LIN {X 0,Y 523.953,Z 186.844,A -85,B 0,C 180,E1 -4818.69,E2 -4818.69} C_VEL
LIN {X 0,Y 523.915,Z 186.845,A -85,B 0,C 180,E1 -4821.08,E2 -4821.08} C_VEL
LIN {X 0,Y 523.898,Z 186.847,A -85,B 0,C 180,E1 -4823.825,E2 -4823.825} C_VEL
LIN {X 0,Y 523.938,Z 186.841,A -85,B 0,C 180,E1 -4826.635,E2 -4826.635} C_VEL
LIN {X 0,Y 523.953,Z 186.839,A -85,B 0,C 180,E1 -4829.356,E2 -4829.356} C_VEL
LIN {X 0,Y 523.973,Z 186.838,A -85,B 0,C 180,E1 -4832.282,E2 -4832.282} C_VEL
LIN {X 0,Y 523.945,Z 186.843,A -85,B 0,C 180,E1 -4834.581,E2 -4834.581} C_VEL
LIN {X 0,Y 523.916,Z 186.848,A -85,B 0,C 180,E1 -4837.756,E2 -4837.756} C_VEL
LIN {X 0,Y 523.971,Z 186.842,A -85,B 0,C 180,E1 -4840.408,E2 -4840.408} C_VEL
LIN {X 0,Y 523.96,Z 186.838,A -85,B 0,C 180,E1 -4842.837,E2 -4842.837} C_VEL
LIN {X 0,Y 523.974,Z 186.837,A -85,B 0,C 180,E1 -4845.236,E2 -4845.236} C_VEL
LIN {X 0,Y 524.009,Z 186.835,A -85,B 0,C 180,E1 -4848.394,E2 -4848.394} C_VEL
LIN {X 0,Y 524,Z 186.836,A -85,B 0,C 180,E1 -4851.516,E2 -4851.516} C_VEL
LIN {X 0,Y 524.078,Z 186.821,A -85,B 0,C 180,E1 -4854.614,E2 -4854.614} C_VEL
LIN {X 0,Y 524.107,Z 186.827,A -85,B 0,C 180,E1 -4857.695,E2 -4857.695} C_VEL
LIN {X 0,Y 524.12,Z 186.819,A -85,B 0,C 180,E1 -4860.768,E2 -4860.768} C_VEL
LIN {X 0,Y 524.07,Z 186.826,A -85,B 0,C 180,E1 -4863.075,E2 -4863.075} C_VEL
LIN {X 0,Y 524.043,Z 186.829,A -85,B 0,C 180,E1 -4866.159,E2 -4866.159} C_VEL
LIN {X 0,Y 523.996,Z 186.84,A -85,B 0,C 180,E1 -4869.262,E2 -4869.262} C_VEL
LIN {X 0,Y 524,Z 186.835,A -85,B 0,C 180,E1 -4871.74,E2 -4871.74} C_VEL
LIN {X 0,Y 523.991,Z 186.841,A -85,B 0,C 180,E1 -4875.053,E2 -4875.053} C_VEL
LIN {X 0,Y 523.962,Z 186.839,A -85,B 0,C 180,E1 -4877.969,E2 -4877.969} C_VEL
LIN {X 0,Y 523.97,Z 186.836,A -85,B 0,C 180,E1 -4880.41,E2 -4880.41} C_VEL
LIN {X 0,Y 523.909,Z 186.851,A -85,B 0,C 180,E1 -4882.894,E2 -4882.894} C_VEL
LIN {X 0,Y 523.951,Z 186.843,A -85,B 0,C 180,E1 -4885.419,E2 -4885.419} C_VEL
LIN {X 0,Y 523.966,Z 186.832,A -85,B 0,C 180,E1 -4887.999,E2 -4887.999} C_VEL
LIN {X 0,Y 523.943,Z 186.846,A -85,B 0,C 180,E1 -4890.855,E2 -4890.855} C_VEL
LIN {X 0,Y 523.96,Z 186.835,A -85,B 0,C 180,E1 -4893.735,E2 -4893.735} C_VEL
LIN {X 0,Y 523.922,Z 186.845,A -85,B 0,C 180,E1 -4896.405,E2 -4896.405} C_VEL
LIN {X 0,Y 523.919,Z 186.842,A -85,B 0,C 180,E1 -4899.085,E2 -4899.085} C_VEL
LIN {X 0,Y 523.951,Z 186.843,A -85,B 0,C 180,E1 -4902.119,E2 -4902.119} C_VEL
LIN {X 0,Y 523.946,Z 186.841,A -85,B 0,C 180,E1 -4905.31,E2 -4905.31} C_VEL
LIN {X 0,Y 523.917,Z 186.845,A -85,B 0,C 180,E1 -4906.914,E2 -4906.914} C_VEL
LIN {X 0,Y 523.253,Z 186.926,A -85,B 0,C 180,E1 -4907.556,E2 -4907.556} C_VEL
LIN {X 0,Y 520.411,Z 187.287,A -85,B 0,C 180,E1 -4908.597,E2 -4908.597} C_VEL
LIN {X 0,Y 518.006,Z 187.591,A -85,B 0,C 180,E1 -4909.436,E2 -4909.436} C_VEL
LIN {X 0,Y 516.969,Z 187.718,A -85,B 0,C 180,E1 -4910.084,E2 -4910.084} C_VEL
LIN {X 0,Y 516.881,Z 187.727,A -85,B 0,C 180,E1 -4910.303,E2 -4910.303} C_VEL
LIN {X 0,Y 516.88,Z 187.72,A -85,B 0,C 180,E1 -4913.343,E2 -4913.343} C_VEL
LIN {X 0,Y 516.912,Z 187.715,A -85,B 0,C 180,E1 -4916.121,E2 -4916.121} C_VEL
LIN {X 0,Y 516.893,Z 187.722,A -85,B 0,C 180,E1 -4918.936,E2 -4918.936} C_VEL
LIN {X 0,Y 516.864,Z 187.729,A -85,B 0,C 180,E1 -4921.582,E2 -4921.582} C_VEL
LIN {X 0,Y 516.931,Z 187.951,A -85,B 0,C 180,E1 -4922.974,E2 -4922.974} C_VEL
LIN {X 0,Y 519.733,Z 200.118,A -85,B 0,C 180,E1 -4924.958,E2 -4924.958} C_VEL
LIN {X 0,Y 519.555,Z 209.088,A -85,B 0,C 180,E1 -4926.27,E2 -4926.27} C_VEL
LIN {X 0,Y 518.755,Z 230.793,A -85,B 0,C 180,E1 -4929.375,E2 -4929.375} C_VEL
LIN {X 0,Y 518.392,Z 244.374,A -85,B 0,C 180,E1 -4931.264,E2 -4931.264} C_VEL
LIN {X 0,Y 520.841,Z 257.475,A -85,B 0,C 180,E1 -4931.568,E2 -4931.568} C_VEL
LIN {X 0,Y 520.186,Z 383.262,A -85,B 0,C 180,E1 -4933.29,E2 -4933.29} C_VEL
LIN {X 0,Y 519.944,Z 397.944,A -85,B 0,C 180,E1 -4933.652,E2 -4933.652} C_VEL
LIN {X 0,Y 519.646,Z 411.088,A -85,B 0,C 180,E1 -4934.131,E2 -4934.131} C_VEL
LIN {X 0,Y 519.251,Z 424.666,A -85,B 0,C 180,E1 -4934.797,E2 -4934.797} C_VEL
LIN {X 0,Y 518.721,Z 437.26,A -85,B 0,C 180,E1 -4935.584,E2 -4935.584} C_VEL
LIN {X 0,Y 518.328,Z 448.694,A -85,B 0,C 180,E1 -4936.474,E2 -4936.474} C_VEL
LIN {X 0,Y 517.874,Z 459.183,A -85,B 0,C 180,E1 -4937.459,E2 -4937.459} C_VEL
LIN {X 0,Y 517.46,Z 469.589,A -85,B 0,C 180,E1 -4938.642,E2 -4938.642} C_VEL
LIN {X 0,Y 517.091,Z 478.189,A -85,B 0,C 180,E1 -4939.823,E2 -4939.823} C_VEL
LIN {X 0,Y 516.781,Z 486.445,A -85,B 0,C 180,E1 -4941.199,E2 -4941.199} C_VEL
LIN {X 0,Y 516.571,Z 493.107,A -85,B 0,C 180,E1 -4942.574,E2 -4942.574} C_VEL
LIN {X 0,Y 516.504,Z 497.705,A -85,B 0,C 180,E1 -4943.75,E2 -4943.75} C_VEL
LIN {X 0,Y 516.312,Z 502.484,A -85,B 0,C 180,E1 -4945.315,E2 -4945.315} C_VEL
LIN {X 0,Y 516.357,Z 505.807,A -85,B 0,C 180,E1 -4946.879,E2 -4946.879} C_VEL
LIN {X 0,Y 516.191,Z 507.794,A -85,B 0,C 180,E1 -4948.439,E2 -4948.439} C_VEL
LIN {X 0,Y 516.166,Z 508.48,A -85,B 0,C 180,E1 -4950,E2 -4950} C_VEL
LIN {X 0,Y 516.189,Z 507.88,A -85,B 0,C 180,E1 -4951.56,E2 -4951.56} C_VEL
LIN {X 0,Y 516.356,Z 505.975,A -85,B 0,C 180,E1 -4953.121,E2 -4953.121} C_VEL
LIN {X 0,Y 516.311,Z 502.723,A -85,B 0,C 180,E1 -4954.684,E2 -4954.684} C_VEL
LIN {X 0,Y 516.502,Z 498.019,A -85,B 0,C 180,E1 -4956.249,E2 -4956.249} C_VEL
LIN {X 0,Y 516.599,Z 491.746,A -85,B 0,C 180,E1 -4957.819,E2 -4957.819} C_VEL
LIN {X 0,Y 516.828,Z 484.765,A -85,B 0,C 180,E1 -4959.194,E2 -4959.194} C_VEL
LIN {X 0,Y 517.185,Z 476.143,A -85,B 0,C 180,E1 -4960.57,E2 -4960.57} C_VEL
LIN {X 0,Y 517.563,Z 467.127,A -85,B 0,C 180,E1 -4961.752,E2 -4961.752} C_VEL
LIN {X 0,Y 517.889,Z 458.139,A -85,B 0,C 180,E1 -4962.739,E2 -4962.739} C_VEL
LIN {X 0,Y 518.339,Z 447.432,A -85,B 0,C 180,E1 -4963.725,E2 -4963.725} C_VEL
LIN {X 0,Y 518.789,Z 435.723,A -85,B 0,C 180,E1 -4964.614,E2 -4964.614} C_VEL
LIN {X 0,Y 519.285,Z 422.762,A -85,B 0,C 180,E1 -4965.402,E2 -4965.402} C_VEL
LIN {X 0,Y 519.719,Z 409.76,A -85,B 0,C 180,E1 -4966.014,E2 -4966.014} C_VEL
LIN {X 0,Y 519.993,Z 396.813,A -85,B 0,C 180,E1 -4966.472,E2 -4966.472} C_VEL
LIN {X 0,Y 520.192,Z 382.646,A -85,B 0,C 180,E1 -4966.81,E2 -4966.81} C_VEL
LIN {X 0,Y 520.805,Z 261.865,A -85,B 0,C 180,E1 -4968.461,E2 -4968.461} C_VEL
LIN {X 0,Y 520.611,Z 255.697,A -85,B 0,C 180,E1 -4968.554,E2 -4968.554} C_VEL
LIN {X 0,Y 518.438,Z 244.638,A -85,B 0,C 180,E1 -4968.809,E2 -4968.809} C_VEL
LIN {X 0,Y 518.502,Z 238.716,A -85,B 0,C 180,E1 -4969.601,E2 -4969.601} C_VEL
LIN {X 0,Y 519.191,Z 218.613,A -85,B 0,C 180,E1 -4972.453,E2 -4972.453} C_VEL
LIN {X 0,Y 519.801,Z 200.601,A -85,B 0,C 180,E1 -4975.058,E2 -4975.058} C_VEL
LIN {X 0,Y 516.902,Z 187.815,A -85,B 0,C 180,E1 -4977.163,E2 -4977.163} C_VEL
LIN {X 0,Y 516.89,Z 187.718,A -85,B 0,C 180,E1 -4980.203,E2 -4980.203} C_VEL
LIN {X 0,Y 516.894,Z 187.715,A -85,B 0,C 180,E1 -4982.946,E2 -4982.946} C_VEL
LIN {X 0,Y 516.887,Z 187.726,A -85,B 0,C 180,E1 -4985.778,E2 -4985.778} C_VEL
LIN {X 0,Y 516.878,Z 187.721,A -85,B 0,C 180,E1 -4988.715,E2 -4988.715} C_VEL
LIN {X 0,Y 516.911,Z 187.72,A -85,B 0,C 180,E1 -4991.774,E2 -4991.774} C_VEL
LIN {X 0,Y 516.919,Z 187.719,A -85,B 0,C 180,E1 -4995.009,E2 -4995.009} C_VEL
LIN {X 0,Y 516.913,Z 187.718,A -85,B 0,C 180,E1 -4998.398,E2 -4998.398} C_VEL
LIN {X 0,Y 516.877,Z 187.724,A -85,B 0,C 180,E1 -5001.283,E2 -5001.283} C_VEL
LIN {X 0,Y 516.886,Z 187.718,A -85,B 0,C 180,E1 -5004.221,E2 -5004.221} C_VEL
LIN {X 0,Y 516.891,Z 187.722,A -85,B 0,C 180,E1 -5007.053,E2 -5007.053} C_VEL
LIN {X 0,Y 516.896,Z 187.716,A -85,B 0,C 180,E1 -5009.796,E2 -5009.796} C_VEL
LIN {X 0,Y 516.923,Z 187.71,A -85,B 0,C 180,E1 -5012.467,E2 -5012.467} C_VEL
LIN {X 0,Y 516.904,Z 187.725,A -85,B 0,C 180,E1 -5015.071,E2 -5015.071} C_VEL
LIN {X 0,Y 516.863,Z 187.724,A -85,B 0,C 180,E1 -5017.621,E2 -5017.621} C_VEL
LIN {X 0,Y 516.926,Z 187.713,A -85,B 0,C 180,E1 -5020.129,E2 -5020.129} C_VEL
LIN {X 0,Y 516.925,Z 187.721,A -85,B 0,C 180,E1 -5022.596,E2 -5022.596} C_VEL
LIN {X 0,Y 516.935,Z 187.719,A -85,B 0,C 180,E1 -5025.03,E2 -5025.03} C_VEL
LIN {X 0,Y 516.958,Z 187.712,A -85,B 0,C 180,E1 -5028.233,E2 -5028.233} C_VEL
LIN {X 0,Y 516.963,Z 187.71,A -85,B 0,C 180,E1 -5031.399,E2 -5031.399} C_VEL
LIN {X 0,Y 517.003,Z 187.705,A -85,B 0,C 180,E1 -5033.757,E2 -5033.757} C_VEL
LIN {X 0,Y 517.077,Z 187.695,A -85,B 0,C 180,E1 -5037.663,E2 -5037.663} C_VEL
LIN {X 0,Y 517.087,Z 187.695,A -85,B 0,C 180,E1 -5040.779,E2 -5040.779} C_VEL
LIN {X 0,Y 517.008,Z 187.705,A -85,B 0,C 180,E1 -5043.117,E2 -5043.117} C_VEL
LIN {X 0,Y 517.004,Z 187.71,A -85,B 0,C 180,E1 -5046.243,E2 -5046.243} C_VEL
LIN {X 0,Y 516.947,Z 187.711,A -85,B 0,C 180,E1 -5049.389,E2 -5049.389} C_VEL
LIN {X 0,Y 516.944,Z 187.717,A -85,B 0,C 180,E1 -5051.807,E2 -5051.807} C_VEL
LIN {X 0,Y 516.936,Z 187.713,A -85,B 0,C 180,E1 -5055.147,E2 -5055.147} C_VEL
LIN {X 0,Y 516.918,Z 187.721,A -85,B 0,C 180,E1 -5058.222,E2 -5058.222} C_VEL
LIN {X 0,Y 516.905,Z 187.717,A -85,B 0,C 180,E1 -5060.702,E2 -5060.702} C_VEL
LIN {X 0,Y 516.904,Z 187.721,A -85,B 0,C 180,E1 -5064.072,E2 -5064.072} C_VEL
LIN {X 0,Y 516.921,Z 187.706,A -85,B 0,C 180,E1 -5066.658,E2 -5066.658} C_VEL
LIN {X 0,Y 516.903,Z 187.724,A -85,B 0,C 180,E1 -5069.524,E2 -5069.524} C_VEL
LIN {X 0,Y 516.891,Z 187.711,A -85,B 0,C 180,E1 -5072.544,E2 -5072.544} C_VEL
LIN {X 0,Y 516.874,Z 187.728,A -85,B 0,C 180,E1 -5075.332,E2 -5075.332} C_VEL
LIN {X 0,Y 516.875,Z 187.722,A -85,B 0,C 180,E1 -5077.944,E2 -5077.944} C_VEL
LIN {X 0,Y 516.877,Z 187.723,A -85,B 0,C 180,E1 -5080.742,E2 -5080.742} C_VEL
LIN {X 0,Y 516.876,Z 187.721,A -85,B 0,C 180,E1 -5082.832,E2 -5082.832} C_VEL
LIN {X 0,Y 516.889,Z 187.725,A -85,B 0,C 180,E1 -5085.007,E2 -5085.007} C_VEL
LIN {X 0,Y 516.908,Z 187.717,A -85,B 0,C 180,E1 -5088.399,E2 -5088.399} C_VEL
LIN {X 0,Y 516.873,Z 187.719,A -85,B 0,C 180,E1 -5091.284,E2 -5091.284} C_VEL
LIN {X 0,Y 516.866,Z 187.719,A -85,B 0,C 180,E1 -5094.22,E2 -5094.22} C_VEL
LIN {X 0,Y 516.877,Z 187.725,A -85,B 0,C 180,E1 -5097.053,E2 -5097.053} C_VEL
LIN {X 0,Y 516.857,Z 187.678,A -85,B 0,C 180,E1 -5099.795,E2 -5099.795} C_VEL
LIN {X 0,Y 516.926,Z 187.879,A -85,B 0,C 180,E1 -5101.392,E2 -5101.392} C_VEL
LIN {X 0,Y 520.508,Z 201.805,A -85,B 0,C 180,E1 -5103.314,E2 -5103.314} C_VEL
LIN {X 0,Y 520.721,Z 205.507,A -85,B 0,C 180,E1 -5103.768,E2 -5103.768} C_VEL
LIN {X 0,Y 519.625,Z 234.25,A -85,B 0,C 180,E1 -5107.118,E2 -5107.118} C_VEL
LIN {X 0,Y 519.292,Z 245.134,A -85,B 0,C 180,E1 -5108.345,E2 -5108.345} C_VEL
LIN {X 0,Y 521.579,Z 259.663,A -85,B 0,C 180,E1 -5108.666,E2 -5108.666} C_VEL
LIN {X 0,Y 520.369,Z 411.25,A -85,B 0,C 180,E1 -5110.871,E2 -5110.871} C_VEL
LIN {X 0,Y 520.061,Z 427.069,A -85,B 0,C 180,E1 -5111.265,E2 -5111.265} C_VEL
LIN {X 0,Y 519.736,Z 441.63,A -85,B 0,C 180,E1 -5111.784,E2 -5111.784} C_VEL
LIN {X 0,Y 519.225,Z 456.376,A -85,B 0,C 180,E1 -5112.473,E2 -5112.473} C_VEL
LIN {X 0,Y 518.806,Z 469.902,A -85,B 0,C 180,E1 -5113.27,E2 -5113.27} C_VEL
LIN {X 0,Y 518.308,Z 483.631,A -85,B 0,C 180,E1 -5114.265,E2 -5114.265} C_VEL
LIN {X 0,Y 517.839,Z 496.096,A -85,B 0,C 180,E1 -5115.359,E2 -5115.359} C_VEL
LIN {X 0,Y 517.44,Z 506.568,A -85,B 0,C 180,E1 -5116.45,E2 -5116.45} C_VEL
LIN {X 0,Y 517.045,Z 517.733,A -85,B 0,C 180,E1 -5117.838,E2 -5117.838} C_VEL
LIN {X 0,Y 516.819,Z 526.971,A -85,B 0,C 180,E1 -5119.224,E2 -5119.224} C_VEL
LIN {X 0,Y 516.55,Z 534.62,A -85,B 0,C 180,E1 -5120.604,E2 -5120.604} C_VEL
LIN {X 0,Y 516.443,Z 541.759,A -85,B 0,C 180,E1 -5122.179,E2 -5122.179} C_VEL
LIN {X 0,Y 516.36,Z 547.363,A -85,B 0,C 180,E1 -5123.749,E2 -5123.749} C_VEL
LIN {X 0,Y 516.374,Z 549.645,A -85,B 0,C 180,E1 -5124.533,E2 -5124.533} C_VEL
LIN {X 0,Y 516.307,Z 553.23,A -85,B 0,C 180,E1 -5126.098,E2 -5126.098} C_VEL
LIN {X 0,Y 516.258,Z 555.585,A -85,B 0,C 180,E1 -5127.66,E2 -5127.66} C_VEL
LIN {X 0,Y 516.157,Z 556.764,A -85,B 0,C 180,E1 -5129.22,E2 -5129.22} C_VEL
LIN {X 0,Y 516.158,Z 556.763,A -85,B 0,C 180,E1 -5130.78,E2 -5130.78} C_VEL
LIN {X 0,Y 516.258,Z 555.58,A -85,B 0,C 180,E1 -5132.341,E2 -5132.341} C_VEL
LIN {X 0,Y 516.307,Z 553.225,A -85,B 0,C 180,E1 -5133.903,E2 -5133.903} C_VEL
LIN {X 0,Y 516.374,Z 549.645,A -85,B 0,C 180,E1 -5135.467,E2 -5135.467} C_VEL
LIN {X 0,Y 516.396,Z 544.743,A -85,B 0,C 180,E1 -5137.036,E2 -5137.036} C_VEL
LIN {X 0,Y 516.514,Z 538.389,A -85,B 0,C 180,E1 -5138.608,E2 -5138.608} C_VEL
LIN {X 0,Y 516.699,Z 530.4,A -85,B 0,C 180,E1 -5140.185,E2 -5140.185} C_VEL
LIN {X 0,Y 516.915,Z 522.234,A -85,B 0,C 180,E1 -5141.517,E2 -5141.517} C_VEL
LIN {X 0,Y 517.199,Z 513.193,A -85,B 0,C 180,E1 -5142.757,E2 -5142.757} C_VEL
LIN {X 0,Y 517.58,Z 502.929,A -85,B 0,C 180,E1 -5143.947,E2 -5143.947} C_VEL
LIN {X 0,Y 518,Z 491.056,A -85,B 0,C 180,E1 -5145.106,E2 -5145.106} C_VEL
LIN {X 0,Y 518.467,Z 478.419,A -85,B 0,C 180,E1 -5146.134,E2 -5146.134} C_VEL
LIN {X 0,Y 518.9,Z 465.073,A -85,B 0,C 180,E1 -5147.031,E2 -5147.031} C_VEL
LIN {X 0,Y 519.391,Z 451.396,A -85,B 0,C 180,E1 -5147.776,E2 -5147.776} C_VEL
LIN {X 0,Y 519.85,Z 436.725,A -85,B 0,C 180,E1 -5148.405,E2 -5148.405} C_VEL
LIN {X 0,Y 520.174,Z 422.03,A -85,B 0,C 180,E1 -5148.876,E2 -5148.876} C_VEL
LIN {X 0,Y 520.43,Z 406.572,A -85,B 0,C 180,E1 -5149.21,E2 -5149.21} C_VEL
LIN {X 0,Y 521.524,Z 258.21,A -85,B 0,C 180,E1 -5151.357,E2 -5151.357} C_VEL
LIN {X 0,Y 519.277,Z 244.941,A -85,B 0,C 180,E1 -5151.668,E2 -5151.668} C_VEL
LIN {X 0,Y 520.013,Z 223.524,A -85,B 0,C 180,E1 -5154.131,E2 -5154.131} C_VEL
LIN {X 0,Y 520.77,Z 203.694,A -85,B 0,C 180,E1 -5156.446,E2 -5156.446} C_VEL
LIN {X 0,Y 519.83,Z 199.121,A -85,B 0,C 180,E1 -5157.044,E2 -5157.044} C_VEL
LIN {X 0,Y 516.929,Z 187.877,A -85,B 0,C 180,E1 -5158.608,E2 -5158.608} C_VEL
LIN {X 0,Y 516.885,Z 187.686,A -85,B 0,C 180,E1 -5161.11,E2 -5161.11} C_VEL
LIN {X 0,Y 516.884,Z 187.722,A -85,B 0,C 180,E1 -5163.962,E2 -5163.962} C_VEL
LIN {X 0,Y 516.875,Z 187.724,A -85,B 0,C 180,E1 -5166.746,E2 -5166.746} C_VEL
LIN {X 0,Y 516.869,Z 187.707,A -85,B 0,C 180,E1 -5169.722,E2 -5169.722} C_VEL
LIN {X 0,Y 516.91,Z 187.717,A -85,B 0,C 180,E1 -5171.775,E2 -5171.775} C_VEL
LIN {X 0,Y 516.893,Z 187.725,A -85,B 0,C 180,E1 -5175.007,E2 -5175.007} C_VEL
LIN {X 0,Y 516.911,Z 187.718,A -85,B 0,C 180,E1 -5178.399,E2 -5178.399} C_VEL
LIN {X 0,Y 516.878,Z 187.72,A -85,B 0,C 180,E1 -5181.284,E2 -5181.284} C_VEL
LIN {X 0,Y 516.868,Z 187.726,A -85,B 0,C 180,E1 -5184.22,E2 -5184.22} C_VEL
LIN {X 0,Y 516.892,Z 187.713,A -85,B 0,C 180,E1 -5187.053,E2 -5187.053} C_VEL
LIN {X 0,Y 516.888,Z 187.721,A -85,B 0,C 180,E1 -5189.796,E2 -5189.796} C_VEL
LIN {X 0,Y 516.923,Z 187.712,A -85,B 0,C 180,E1 -5192.467,E2 -5192.467} C_VEL
LIN {X 0,Y 516.873,Z 187.72,A -85,B 0,C 180,E1 -5195.07,E2 -5195.07} C_VEL
LIN {X 0,Y 516.865,Z 187.725,A -85,B 0,C 180,E1 -5197.621,E2 -5197.621} C_VEL
LIN {X 0,Y 516.928,Z 187.723,A -85,B 0,C 180,E1 -5200.13,E2 -5200.13} C_VEL
LIN {X 0,Y 516.924,Z 187.716,A -85,B 0,C 180,E1 -5202.596,E2 -5202.596} C_VEL
LIN {X 0,Y 516.939,Z 187.713,A -85,B 0,C 180,E1 -5205.03,E2 -5205.03} C_VEL
LIN {X 0,Y 516.963,Z 187.715,A -85,B 0,C 180,E1 -5208.234,E2 -5208.234} C_VEL
LIN {X 0,Y 516.965,Z 187.711,A -85,B 0,C 180,E1 -5211.4,E2 -5211.4} C_VEL
LIN {X 0,Y 517.007,Z 187.71,A -85,B 0,C 180,E1 -5213.757,E2 -5213.757} C_VEL
LIN {X 0,Y 517.08,Z 187.702,A -85,B 0,C 180,E1 -5217.663,E2 -5217.663} C_VEL
LIN {X 0,Y 517.09,Z 187.695,A -85,B 0,C 180,E1 -5220.779,E2 -5220.779} C_VEL
LIN {X 0,Y 517.011,Z 187.705,A -85,B 0,C 180,E1 -5223.117,E2 -5223.117} C_VEL
LIN {X 0,Y 517.007,Z 187.705,A -85,B 0,C 180,E1 -5226.243,E2 -5226.243} C_VEL
LIN {X 0,Y 516.951,Z 187.72,A -85,B 0,C 180,E1 -5229.389,E2 -5229.389} C_VEL
LIN {X 0,Y 516.949,Z 187.713,A -85,B 0,C 180,E1 -5231.807,E2 -5231.807} C_VEL
LIN {X 0,Y 516.942,Z 187.72,A -85,B 0,C 180,E1 -5235.147,E2 -5235.147} C_VEL
LIN {X 0,Y 516.923,Z 187.716,A -85,B 0,C 180,E1 -5238.222,E2 -5238.222} C_VEL
LIN {X 0,Y 516.91,Z 187.717,A -85,B 0,C 180,E1 -5240.702,E2 -5240.702} C_VEL
LIN {X 0,Y 516.901,Z 187.716,A -85,B 0,C 180,E1 -5244.073,E2 -5244.073} C_VEL
LIN {X 0,Y 516.922,Z 187.72,A -85,B 0,C 180,E1 -5246.658,E2 -5246.658} C_VEL
LIN {X 0,Y 516.909,Z 187.715,A -85,B 0,C 180,E1 -5249.524,E2 -5249.524} C_VEL
LIN {X 0,Y 516.894,Z 187.724,A -85,B 0,C 180,E1 -5252.544,E2 -5252.544} C_VEL
LIN {X 0,Y 516.882,Z 187.719,A -85,B 0,C 180,E1 -5255.333,E2 -5255.333} C_VEL
LIN {X 0,Y 516.88,Z 187.722,A -85,B 0,C 180,E1 -5257.943,E2 -5257.943} C_VEL
LIN {X 0,Y 516.882,Z 187.724,A -85,B 0,C 180,E1 -5260.742,E2 -5260.742} C_VEL
LIN {X 0,Y 516.882,Z 187.724,A -85,B 0,C 180,E1 -5262.832,E2 -5262.832} C_VEL
LIN {X 0,Y 516.923,Z 187.719,A -85,B 0,C 180,E1 -5265.01,E2 -5265.01} C_VEL
LIN {X 0,Y 516.916,Z 187.72,A -85,B 0,C 180,E1 -5268.399,E2 -5268.399} C_VEL
LIN {X 0,Y 516.881,Z 187.727,A -85,B 0,C 180,E1 -5270.303,E2 -5270.303} C_VEL
LIN {X 0,Y 516.21,Z 187.807,A -85,B 0,C 180,E1 -5270.953,E2 -5270.953} C_VEL
LIN {X 0,Y 513.363,Z 188.163,A -85,B 0,C 180,E1 -5272.009,E2 -5272.009} C_VEL
LIN {X 0,Y 510.954,Z 188.46,A -85,B 0,C 180,E1 -5272.859,E2 -5272.859} C_VEL
LIN {X 0,Y 509.913,Z 188.588,A -85,B 0,C 180,E1 -5273.516,E2 -5273.516} C_VEL
LIN {X 0,Y 509.824,Z 188.6,A -85,B 0,C 180,E1 -5273.738,E2 -5273.738} C_VEL
LIN {X 0,Y 509.862,Z 188.589,A -85,B 0,C 180,E1 -5276.539,E2 -5276.539} C_VEL
LIN {X 0,Y 509.847,Z 188.599,A -85,B 0,C 180,E1 -5279.334,E2 -5279.334} C_VEL
LIN {X 0,Y 509.871,Z 188.59,A -85,B 0,C 180,E1 -5282.499,E2 -5282.499} C_VEL
LIN {X 0,Y 509.907,Z 189.025,A -85,B 0,C 180,E1 -5282.724,E2 -5282.724} C_VEL
LIN {X 0,Y 512.941,Z 201.979,A -85,B 0,C 180,E1 -5284.866,E2 -5284.866} C_VEL
LIN {X 0,Y 512.535,Z 214.705,A -85,B 0,C 180,E1 -5286.74,E2 -5286.74} C_VEL
LIN {X 0,Y 511.72,Z 236.742,A -85,B 0,C 180,E1 -5289.919,E2 -5289.919} C_VEL
LIN {X 0,Y 511.525,Z 244.588,A -85,B 0,C 180,E1 -5290.994,E2 -5290.994} C_VEL
LIN {X 0,Y 514.172,Z 258.182,A -85,B 0,C 180,E1 -5291.307,E2 -5291.307} C_VEL
LIN {X 0,Y 513.489,Z 384.022,A -85,B 0,C 180,E1 -5293.04,E2 -5293.04} C_VEL
LIN {X 0,Y 513.247,Z 398.289,A -85,B 0,C 180,E1 -5293.399,E2 -5293.399} C_VEL
LIN {X 0,Y 512.891,Z 412.102,A -85,B 0,C 180,E1 -5293.912,E2 -5293.912} C_VEL
LIN {X 0,Y 512.552,Z 423.868,A -85,B 0,C 180,E1 -5294.492,E2 -5294.492} C_VEL
LIN {X 0,Y 511.992,Z 436.682,A -85,B 0,C 180,E1 -5295.289,E2 -5295.289} C_VEL
LIN {X 0,Y 511.511,Z 448.28,A -85,B 0,C 180,E1 -5296.188,E2 -5296.188} C_VEL
LIN {X 0,Y 510.987,Z 459.837,A -85,B 0,C 180,E1 -5297.287,E2 -5297.287} C_VEL
LIN {X 0,Y 510.52,Z 470.169,A -85,B 0,C 180,E1 -5298.486,E2 -5298.486} C_VEL
LIN {X 0,Y 510.13,Z 478.708,A -85,B 0,C 180,E1 -5299.683,E2 -5299.683} C_VEL
LIN {X 0,Y 509.781,Z 486.911,A -85,B 0,C 180,E1 -5301.077,E2 -5301.077} C_VEL
LIN {X 0,Y 509.546,Z 493.532,A -85,B 0,C 180,E1 -5302.471,E2 -5302.471} C_VEL
LIN {X 0,Y 509.413,Z 499.453,A -85,B 0,C 180,E1 -5304.061,E2 -5304.061} C_VEL
LIN {X 0,Y 509.231,Z 502.855,A -85,B 0,C 180,E1 -5305.25,E2 -5305.25} C_VEL
LIN {X 0,Y 509.281,Z 506.157,A -85,B 0,C 180,E1 -5306.835,E2 -5306.835} C_VEL
LIN {X 0,Y 509.111,Z 508.132,A -85,B 0,C 180,E1 -5308.418,E2 -5308.418} C_VEL
LIN {X 0,Y 509.076,Z 508.812,A -85,B 0,C 180,E1 -5310,E2 -5310} C_VEL
LIN {X 0,Y 509.11,Z 508.215,A -85,B 0,C 180,E1 -5311.582,E2 -5311.582} C_VEL
LIN {X 0,Y 509.266,Z 506.323,A -85,B 0,C 180,E1 -5313.164,E2 -5313.164} C_VEL
LIN {X 0,Y 509.23,Z 503.09,A -85,B 0,C 180,E1 -5314.75,E2 -5314.75} C_VEL
LIN {X 0,Y 509.465,Z 498.412,A -85,B 0,C 180,E1 -5316.336,E2 -5316.336} C_VEL
LIN {X 0,Y 509.58,Z 492.172,A -85,B 0,C 180,E1 -5317.927,E2 -5317.927} C_VEL
LIN {X 0,Y 509.836,Z 485.229,A -85,B 0,C 180,E1 -5319.321,E2 -5319.321} C_VEL
LIN {X 0,Y 510.223,Z 476.657,A -85,B 0,C 180,E1 -5320.716,E2 -5320.716} C_VEL
LIN {X 0,Y 510.639,Z 467.7,A -85,B 0,C 180,E1 -5321.914,E2 -5321.914} C_VEL
LIN {X 0,Y 511.121,Z 456.852,A -85,B 0,C 180,E1 -5323.113,E2 -5323.113} C_VEL
LIN {X 0,Y 511.602,Z 445.802,A -85,B 0,C 180,E1 -5324.113,E2 -5324.113} C_VEL
LIN {X 0,Y 512.136,Z 433.594,A -85,B 0,C 180,E1 -5325.011,E2 -5325.011} C_VEL
LIN {X 0,Y 512.571,Z 421.835,A -85,B 0,C 180,E1 -5325.711,E2 -5325.711} C_VEL
LIN {X 0,Y 513.004,Z 409.13,A -85,B 0,C 180,E1 -5326.303,E2 -5326.303} C_VEL
LIN {X 0,Y 513.297,Z 395.96,A -85,B 0,C 180,E1 -5326.761,E2 -5326.761} C_VEL
LIN {X 0,Y 513.509,Z 381.878,A -85,B 0,C 180,E1 -5327.087,E2 -5327.087} C_VEL
LIN {X 0,Y 514.144,Z 258.405,A -85,B 0,C 180,E1 -5328.78,E2 -5328.78} C_VEL
LIN {X 0,Y 511.545,Z 244.541,A -85,B 0,C 180,E1 -5329.099,E2 -5329.099} C_VEL
LIN {X 0,Y 511.938,Z 230.922,A -85,B 0,C 180,E1 -5331.009,E2 -5331.009} C_VEL
LIN {X 0,Y 512.728,Z 209.821,A -85,B 0,C 180,E1 -5334.065,E2 -5334.065} C_VEL
LIN {X 0,Y 512.877,Z 201.786,A -85,B 0,C 180,E1 -5335.257,E2 -5335.257} C_VEL
LIN {X 0,Y 509.882,Z 188.697,A -85,B 0,C 180,E1 -5337.444,E2 -5337.444} C_VEL
LIN {X 0,Y 509.844,Z 188.599,A -85,B 0,C 180,E1 -5340.665,E2 -5340.665} C_VEL
LIN {X 0,Y 509.859,Z 188.589,A -85,B 0,C 180,E1 -5343.46,E2 -5343.46} C_VEL
LIN {X 0,Y 509.833,Z 188.599,A -85,B 0,C 180,E1 -5346.352,E2 -5346.352} C_VEL
LIN {X 0,Y 509.831,Z 188.602,A -85,B 0,C 180,E1 -5349.47,E2 -5349.47} C_VEL
LIN {X 0,Y 509.831,Z 188.596,A -85,B 0,C 180,E1 -5352.489,E2 -5352.489} C_VEL
LIN {X 0,Y 509.853,Z 188.6,A -85,B 0,C 180,E1 -5355.331,E2 -5355.331} C_VEL
LIN {X 0,Y 509.855,Z 188.597,A -85,B 0,C 180,E1 -5358.574,E2 -5358.574} C_VEL
LIN {X 0,Y 509.846,Z 188.601,A -85,B 0,C 180,E1 -5361.786,E2 -5361.786} C_VEL
LIN {X 0,Y 509.841,Z 188.596,A -85,B 0,C 180,E1 -5364.623,E2 -5364.623} C_VEL
LIN {X 0,Y 509.858,Z 188.601,A -85,B 0,C 180,E1 -5367.48,E2 -5367.48} C_VEL
LIN {X 0,Y 509.876,Z 188.589,A -85,B 0,C 180,E1 -5370.268,E2 -5370.268} C_VEL
LIN {X 0,Y 509.88,Z 188.593,A -85,B 0,C 180,E1 -5372.944,E2 -5372.944} C_VEL
LIN {X 0,Y 509.863,Z 188.595,A -85,B 0,C 180,E1 -5375.574,E2 -5375.574} C_VEL
LIN {X 0,Y 509.844,Z 188.603,A -85,B 0,C 180,E1 -5378.998,E2 -5378.998} C_VEL
LIN {X 0,Y 509.882,Z 188.593,A -85,B 0,C 180,E1 -5381.999,E2 -5381.999} C_VEL
LIN {X 0,Y 509.903,Z 188.595,A -85,B 0,C 180,E1 -5384.818,E2 -5384.818} C_VEL
LIN {X 0,Y 509.894,Z 188.59,A -85,B 0,C 180,E1 -5388.123,E2 -5388.123} C_VEL
LIN {X 0,Y 509.909,Z 188.589,A -85,B 0,C 180,E1 -5391.28,E2 -5391.28} C_VEL
LIN {X 0,Y 509.971,Z 188.581,A -85,B 0,C 180,E1 -5393.67,E2 -5393.67} C_VEL
LIN {X 0,Y 510.048,Z 188.57,A -85,B 0,C 180,E1 -5397.631,E2 -5397.631} C_VEL
LIN {X 0,Y 510.057,Z 188.57,A -85,B 0,C 180,E1 -5400.789,E2 -5400.789} C_VEL
LIN {X 0,Y 509.95,Z 188.584,A -85,B 0,C 180,E1 -5403.16,E2 -5403.16} C_VEL
LIN {X 0,Y 509.972,Z 188.587,A -85,B 0,C 180,E1 -5406.33,E2 -5406.33} C_VEL
LIN {X 0,Y 509.909,Z 188.589,A -85,B 0,C 180,E1 -5408.72,E2 -5408.72} C_VEL
LIN {X 0,Y 509.896,Z 188.597,A -85,B 0,C 180,E1 -5411.932,E2 -5411.932} C_VEL
LIN {X 0,Y 509.886,Z 188.592,A -85,B 0,C 180,E1 -5415.242,E2 -5415.242} C_VEL
LIN {X 0,Y 509.881,Z 188.597,A -85,B 0,C 180,E1 -5418.001,E2 -5418.001} C_VEL
LIN {X 0,Y 509.843,Z 188.596,A -85,B 0,C 180,E1 -5421.002,E2 -5421.002} C_VEL
LIN {X 0,Y 509.863,Z 188.594,A -85,B 0,C 180,E1 -5424.426,E2 -5424.426} C_VEL
LIN {X 0,Y 509.88,Z 188.584,A -85,B 0,C 180,E1 -5427.056,E2 -5427.056} C_VEL
LIN {X 0,Y 509.85,Z 188.604,A -85,B 0,C 180,E1 -5429.751,E2 -5429.751} C_VEL
LIN {X 0,Y 509.868,Z 188.586,A -85,B 0,C 180,E1 -5432.775,E2 -5432.775} C_VEL
LIN {X 0,Y 509.834,Z 188.605,A -85,B 0,C 180,E1 -5435.581,E2 -5435.581} C_VEL
LIN {X 0,Y 509.844,Z 188.595,A -85,B 0,C 180,E1 -5438.338,E2 -5438.338} C_VEL
LIN {X 0,Y 509.849,Z 188.599,A -85,B 0,C 180,E1 -5441.426,E2 -5441.426} C_VEL
LIN {X 0,Y 509.833,Z 188.601,A -85,B 0,C 180,E1 -5444.67,E2 -5444.67} C_VEL
LIN {X 0,Y 509.85,Z 188.596,A -85,B 0,C 180,E1 -5448.104,E2 -5448.104} C_VEL
LIN {X 0,Y 509.833,Z 188.585,A -85,B 0,C 180,E1 -5450.647,E2 -5450.647} C_VEL
LIN {X 0,Y 509.82,Z 188.598,A -85,B 0,C 180,E1 -5453.647,E2 -5453.647} C_VEL
LIN {X 0,Y 509.837,Z 188.603,A -85,B 0,C 180,E1 -5456.538,E2 -5456.538} C_VEL
LIN {X 0,Y 509.828,Z 188.556,A -85,B 0,C 180,E1 -5459.334,E2 -5459.334} C_VEL
LIN {X 0,Y 509.901,Z 188.758,A -85,B 0,C 180,E1 -5461.088,E2 -5461.088} C_VEL
LIN {X 0,Y 513.696,Z 203.561,A -85,B 0,C 180,E1 -5463.162,E2 -5463.162} C_VEL
LIN {X 0,Y 514.036,Z 205.372,A -85,B 0,C 180,E1 -5463.4,E2 -5463.4} C_VEL
LIN {X 0,Y 512.857,Z 234.031,A -85,B 0,C 180,E1 -5466.792,E2 -5466.792} C_VEL
LIN {X 0,Y 512.462,Z 245.285,A -85,B 0,C 180,E1 -5468.069,E2 -5468.069} C_VEL
LIN {X 0,Y 514.912,Z 260.394,A -85,B 0,C 180,E1 -5468.409,E2 -5468.409} C_VEL
LIN {X 0,Y 513.575,Z 411.141,A -85,B 0,C 180,E1 -5470.646,E2 -5470.646} C_VEL
LIN {X 0,Y 513.254,Z 426.906,A -85,B 0,C 180,E1 -5471.047,E2 -5471.047} C_VEL
LIN {X 0,Y 512.869,Z 441.694,A -85,B 0,C 180,E1 -5471.584,E2 -5471.584} C_VEL
LIN {X 0,Y 512.379,Z 455.418,A -85,B 0,C 180,E1 -5472.231,E2 -5472.231} C_VEL
LIN {X 0,Y 511.89,Z 469.037,A -85,B 0,C 180,E1 -5473.038,E2 -5473.038} C_VEL
LIN {X 0,Y 511.353,Z 482.887,A -85,B 0,C 180,E1 -5474.046,E2 -5474.046} C_VEL
LIN {X 0,Y 510.861,Z 495.432,A -85,B 0,C 180,E1 -5475.154,E2 -5475.154} C_VEL
LIN {X 0,Y 510.381,Z 507.693,A -85,B 0,C 180,E1 -5476.462,E2 -5476.462} C_VEL
LIN {X 0,Y 510.001,Z 517.196,A -85,B 0,C 180,E1 -5477.667,E2 -5477.667} C_VEL
LIN {X 0,Y 509.743,Z 526.491,A -85,B 0,C 180,E1 -5479.072,E2 -5479.072} C_VEL
LIN {X 0,Y 509.476,Z 534.184,A -85,B 0,C 180,E1 -5480.472,E2 -5480.472} C_VEL
LIN {X 0,Y 509.361,Z 541.357,A -85,B 0,C 180,E1 -5482.07,E2 -5482.07} C_VEL
LIN {X 0,Y 509.265,Z 546.985,A -85,B 0,C 180,E1 -5483.662,E2 -5483.662} C_VEL
LIN {X 0,Y 509.158,Z 551.233,A -85,B 0,C 180,E1 -5485.25,E2 -5485.25} C_VEL
LIN {X 0,Y 509.188,Z 554.212,A -85,B 0,C 180,E1 -5486.835,E2 -5486.835} C_VEL
LIN {X 0,Y 509.11,Z 555.983,A -85,B 0,C 180,E1 -5488.418,E2 -5488.418} C_VEL
LIN {X 0,Y 509.064,Z 556.587,A -85,B 0,C 180,E1 -5490,E2 -5490} C_VEL
LIN {X 0,Y 509.11,Z 555.98,A -85,B 0,C 180,E1 -5491.582,E2 -5491.582} C_VEL
LIN {X 0,Y 509.188,Z 554.206,A -85,B 0,C 180,E1 -5493.165,E2 -5493.165} C_VEL
LIN {X 0,Y 509.158,Z 551.229,A -85,B 0,C 180,E1 -5494.751,E2 -5494.751} C_VEL
LIN {X 0,Y 509.306,Z 546.99,A -85,B 0,C 180,E1 -5496.338,E2 -5496.338} C_VEL
LIN {X 0,Y 509.362,Z 541.355,A -85,B 0,C 180,E1 -5497.931,E2 -5497.931} C_VEL
LIN {X 0,Y 509.476,Z 534.175,A -85,B 0,C 180,E1 -5499.528,E2 -5499.528} C_VEL
LIN {X 0,Y 509.739,Z 526.484,A -85,B 0,C 180,E1 -5500.928,E2 -5500.928} C_VEL
LIN {X 0,Y 510.006,Z 517.194,A -85,B 0,C 180,E1 -5502.333,E2 -5502.333} C_VEL
LIN {X 0,Y 510.442,Z 505.946,A -85,B 0,C 180,E1 -5503.739,E2 -5503.739} C_VEL
LIN {X 0,Y 510.918,Z 494.363,A -85,B 0,C 180,E1 -5504.947,E2 -5504.947} C_VEL
LIN {X 0,Y 511.359,Z 482.891,A -85,B 0,C 180,E1 -5505.955,E2 -5505.955} C_VEL
LIN {X 0,Y 511.865,Z 469.024,A -85,B 0,C 180,E1 -5506.964,E2 -5506.964} C_VEL
LIN {X 0,Y 512.407,Z 454.405,A -85,B 0,C 180,E1 -5507.82,E2 -5507.82} C_VEL
LIN {X 0,Y 512.931,Z 439.537,A -85,B 0,C 180,E1 -5508.504,E2 -5508.504} C_VEL
LIN {X 0,Y 513.294,Z 424.558,A -85,B 0,C 180,E1 -5509.024,E2 -5509.024} C_VEL
LIN {X 0,Y 513.601,Z 409.813,A -85,B 0,C 180,E1 -5509.38,E2 -5509.38} C_VEL
LIN {X 0,Y 514.903,Z 259.98,A -85,B 0,C 180,E1 -5511.597,E2 -5511.597} C_VEL
LIN {X 0,Y 512.447,Z 244.964,A -85,B 0,C 180,E1 -5511.948,E2 -5511.948} C_VEL
LIN {X 0,Y 513.202,Z 225.177,A -85,B 0,C 180,E1 -5514.257,E2 -5514.257} C_VEL
LIN {X 0,Y 514.006,Z 205.361,A -85,B 0,C 180,E1 -5516.602,E2 -5516.602} C_VEL
LIN {X 0,Y 510.66,Z 191.731,A -85,B 0,C 180,E1 -5518.465,E2 -5518.465} C_VEL
LIN {X 0,Y 509.891,Z 188.72,A -85,B 0,C 180,E1 -5518.928,E2 -5518.928} C_VEL
LIN {X 0,Y 509.816,Z 188.577,A -85,B 0,C 180,E1 -5521.59,E2 -5521.59} C_VEL
LIN {X 0,Y 509.836,Z 188.597,A -85,B 0,C 180,E1 -5524.414,E2 -5524.414} C_VEL
LIN {X 0,Y 509.814,Z 188.605,A -85,B 0,C 180,E1 -5527.341,E2 -5527.341} C_VEL
LIN {X 0,Y 509.836,Z 188.585,A -85,B 0,C 180,E1 -5530.382,E2 -5530.382} C_VEL
LIN {X 0,Y 509.82,Z 188.605,A -85,B 0,C 180,E1 -5533.062,E2 -5533.062} C_VEL
LIN {X 0,Y 509.82,Z 188.601,A -85,B 0,C 180,E1 -5535.793,E2 -5535.793} C_VEL
LIN {X 0,Y 509.853,Z 188.598,A -85,B 0,C 180,E1 -5538.574,E2 -5538.574} C_VEL
LIN {X 0,Y 509.848,Z 188.595,A -85,B 0,C 180,E1 -5541.786,E2 -5541.786} C_VEL
LIN {X 0,Y 509.828,Z 188.607,A -85,B 0,C 180,E1 -5544.622,E2 -5544.622} C_VEL
LIN {X 0,Y 509.858,Z 188.587,A -85,B 0,C 180,E1 -5547.481,E2 -5547.481} C_VEL
LIN {X 0,Y 509.855,Z 188.603,A -85,B 0,C 180,E1 -5550.274,E2 -5550.274} C_VEL
LIN {X 0,Y 509.881,Z 188.583,A -85,B 0,C 180,E1 -5552.944,E2 -5552.944} C_VEL
LIN {X 0,Y 509.848,Z 188.596,A -85,B 0,C 180,E1 -5555.573,E2 -5555.573} C_VEL
LIN {X 0,Y 509.819,Z 188.606,A -85,B 0,C 180,E1 -5558.149,E2 -5558.149} C_VEL
LIN {X 0,Y 509.86,Z 188.597,A -85,B 0,C 180,E1 -5560.682,E2 -5560.682} C_VEL
LIN {X 0,Y 509.878,Z 188.592,A -85,B 0,C 180,E1 -5563.175,E2 -5563.175} C_VEL
LIN {X 0,Y 509.861,Z 188.599,A -85,B 0,C 180,E1 -5565.634,E2 -5565.634} C_VEL
LIN {X 0,Y 509.91,Z 188.589,A -85,B 0,C 180,E1 -5568.875,E2 -5568.875} C_VEL
LIN {X 0,Y 509.948,Z 188.589,A -85,B 0,C 180,E1 -5572.079,E2 -5572.079} C_VEL
LIN {X 0,Y 509.978,Z 188.578,A -85,B 0,C 180,E1 -5574.464,E2 -5574.464} C_VEL
LIN {X 0,Y 510.051,Z 188.578,A -85,B 0,C 180,E1 -5577.631,E2 -5577.631} C_VEL
LIN {X 0,Y 510.061,Z 188.57,A -85,B 0,C 180,E1 -5580.79,E2 -5580.79} C_VEL
LIN {X 0,Y 509.953,Z 188.585,A -85,B 0,C 180,E1 -5583.16,E2 -5583.16} C_VEL
LIN {X 0,Y 509.975,Z 188.58,A -85,B 0,C 180,E1 -5586.33,E2 -5586.33} C_VEL
LIN {X 0,Y 509.913,Z 188.588,A -85,B 0,C 180,E1 -5588.72,E2 -5588.72} C_VEL
LIN {X 0,Y 509.902,Z 188.589,A -85,B 0,C 180,E1 -5591.932,E2 -5591.932} C_VEL
LIN {X 0,Y 509.892,Z 188.597,A -85,B 0,C 180,E1 -5595.242,E2 -5595.242} C_VEL
LIN {X 0,Y 509.88,Z 188.593,A -85,B 0,C 180,E1 -5597.999,E2 -5597.999} C_VEL
LIN {X 0,Y 509.848,Z 188.601,A -85,B 0,C 180,E1 -5601.002,E2 -5601.002} C_VEL
LIN {X 0,Y 509.862,Z 188.595,A -85,B 0,C 180,E1 -5604.427,E2 -5604.427} C_VEL
LIN {X 0,Y 509.882,Z 188.594,A -85,B 0,C 180,E1 -5607.056,E2 -5607.056} C_VEL
LIN {X 0,Y 509.856,Z 188.592,A -85,B 0,C 180,E1 -5609.751,E2 -5609.751} C_VEL
LIN {X 0,Y 509.872,Z 188.601,A -85,B 0,C 180,E1 -5612.774,E2 -5612.774} C_VEL
LIN {X 0,Y 509.842,Z 188.595,A -85,B 0,C 180,E1 -5615.581,E2 -5615.581} C_VEL
LIN {X 0,Y 509.849,Z 188.601,A -85,B 0,C 180,E1 -5618.338,E2 -5618.338} C_VEL
LIN {X 0,Y 509.854,Z 188.597,A -85,B 0,C 180,E1 -5621.426,E2 -5621.426} C_VEL
LIN {X 0,Y 509.857,Z 188.599,A -85,B 0,C 180,E1 -5624.668,E2 -5624.668} C_VEL
LIN {X 0,Y 509.858,Z 188.596,A -85,B 0,C 180,E1 -5628.103,E2 -5628.103} C_VEL
LIN {X 0,Y 509.846,Z 188.6,A -85,B 0,C 180,E1 -5630.648,E2 -5630.648} C_VEL
LIN {X 0,Y 509.824,Z 188.6,A -85,B 0,C 180,E1 -5633.738,E2 -5633.738} C_VEL
LIN {X 0,Y 509.158,Z 188.691,A -85,B 0,C 180,E1 -5634.398,E2 -5634.398} C_VEL
LIN {X 0,Y 506.344,Z 189.035,A -85,B 0,C 180,E1 -5635.47,E2 -5635.47} C_VEL
LIN {X 0,Y 503.955,Z 189.326,A -85,B 0,C 180,E1 -5636.333,E2 -5636.333} C_VEL
LIN {X 0,Y 502.907,Z 189.454,A -85,B 0,C 180,E1 -5637,E2 -5637} C_VEL
LIN {X 0,Y 502.809,Z 189.466,A -85,B 0,C 180,E1 -5637.225,E2 -5637.225} C_VEL
LIN {X 0,Y 502.816,Z 189.468,A -85,B 0,C 180,E1 -5640.065,E2 -5640.065} C_VEL
LIN {X 0,Y 502.875,Z 189.695,A -85,B 0,C 180,E1 -5642.395,E2 -5642.395} C_VEL
LIN {X 0,Y 506.093,Z 203.615,A -85,B 0,C 180,E1 -5644.733,E2 -5644.733} C_VEL
LIN {X 0,Y 505.9,Z 212.213,A -85,B 0,C 180,E1 -5646.025,E2 -5646.025} C_VEL
LIN {X 0,Y 504.962,Z 234.156,A -85,B 0,C 180,E1 -5649.238,E2 -5649.238} C_VEL
LIN {X 0,Y 504.625,Z 244.422,A -85,B 0,C 180,E1 -5650.69,E2 -5650.69} C_VEL
LIN {X 0,Y 507.536,Z 259.583,A -85,B 0,C 180,E1 -5651.05,E2 -5651.05} C_VEL
LIN {X 0,Y 506.816,Z 384.647,A -85,B 0,C 180,E1 -5652.784,E2 -5652.784} C_VEL
LIN {X 0,Y 506.549,Z 398.703,A -85,B 0,C 180,E1 -5653.142,E2 -5653.142} C_VEL
LIN {X 0,Y 506.193,Z 412.044,A -85,B 0,C 180,E1 -5653.64,E2 -5653.64} C_VEL
LIN {X 0,Y 505.857,Z 423.042,A -85,B 0,C 180,E1 -5654.178,E2 -5654.178} C_VEL
LIN {X 0,Y 505.246,Z 436.105,A -85,B 0,C 180,E1 -5654.985,E2 -5654.985} C_VEL
LIN {X 0,Y 504.718,Z 447.863,A -85,B 0,C 180,E1 -5655.896,E2 -5655.896} C_VEL
LIN {X 0,Y 504.153,Z 458.589,A -85,B 0,C 180,E1 -5656.907,E2 -5656.907} C_VEL
LIN {X 0,Y 503.688,Z 469.169,A -85,B 0,C 180,E1 -5658.123,E2 -5658.123} C_VEL
LIN {X 0,Y 503.23,Z 477.924,A -85,B 0,C 180,E1 -5659.336,E2 -5659.336} C_VEL
LIN {X 0,Y 502.805,Z 486.311,A -85,B 0,C 180,E1 -5660.75,E2 -5660.75} C_VEL
LIN {X 0,Y 502.584,Z 492.213,A -85,B 0,C 180,E1 -5661.961,E2 -5661.961} C_VEL
LIN {X 0,Y 502.402,Z 498.508,A -85,B 0,C 180,E1 -5663.574,E2 -5663.574} C_VEL
LIN {X 0,Y 502.152,Z 503.231,A -85,B 0,C 180,E1 -5665.183,E2 -5665.183} C_VEL
LIN {X 0,Y 502.194,Z 506.51,A -85,B 0,C 180,E1 -5666.791,E2 -5666.791} C_VEL
LIN {X 0,Y 502.035,Z 508.47,A -85,B 0,C 180,E1 -5668.395,E2 -5668.395} C_VEL
LIN {X 0,Y 501.99,Z 509.145,A -85,B 0,C 180,E1 -5670,E2 -5670} C_VEL
LIN {X 0,Y 502.034,Z 508.551,A -85,B 0,C 180,E1 -5671.604,E2 -5671.604} C_VEL
LIN {X 0,Y 502.181,Z 506.672,A -85,B 0,C 180,E1 -5673.209,E2 -5673.209} C_VEL
LIN {X 0,Y 502.151,Z 503.461,A -85,B 0,C 180,E1 -5674.817,E2 -5674.817} C_VEL
LIN {X 0,Y 502.402,Z 498.811,A -85,B 0,C 180,E1 -5676.425,E2 -5676.425} C_VEL
LIN {X 0,Y 502.544,Z 492.607,A -85,B 0,C 180,E1 -5678.039,E2 -5678.039} C_VEL
LIN {X 0,Y 502.841,Z 485.707,A -85,B 0,C 180,E1 -5679.452,E2 -5679.452} C_VEL
LIN {X 0,Y 503.268,Z 477.187,A -85,B 0,C 180,E1 -5680.866,E2 -5680.866} C_VEL
LIN {X 0,Y 503.748,Z 467.136,A -85,B 0,C 180,E1 -5682.226,E2 -5682.226} C_VEL
LIN {X 0,Y 504.288,Z 456.486,A -85,B 0,C 180,E1 -5683.396,E2 -5683.396} C_VEL
LIN {X 0,Y 504.838,Z 445.293,A -85,B 0,C 180,E1 -5684.409,E2 -5684.409} C_VEL
LIN {X 0,Y 505.421,Z 432.895,A -85,B 0,C 180,E1 -5685.319,E2 -5685.319} C_VEL
LIN {X 0,Y 505.829,Z 420.865,A -85,B 0,C 180,E1 -5686.03,E2 -5686.03} C_VEL
LIN {X 0,Y 506.346,Z 406.743,A -85,B 0,C 180,E1 -5686.666,E2 -5686.666} C_VEL
LIN {X 0,Y 506.663,Z 392.828,A -85,B 0,C 180,E1 -5687.117,E2 -5687.117} C_VEL
LIN {X 0,Y 506.863,Z 379.391,A -85,B 0,C 180,E1 -5687.396,E2 -5687.396} C_VEL
LIN {X 0,Y 507.466,Z 260.171,A -85,B 0,C 180,E1 -5689.034,E2 -5689.034} C_VEL
LIN {X 0,Y 507.019,Z 256.502,A -85,B 0,C 180,E1 -5689.105,E2 -5689.105} C_VEL
LIN {X 0,Y 504.637,Z 244.319,A -85,B 0,C 180,E1 -5689.407,E2 -5689.407} C_VEL
LIN {X 0,Y 505.335,Z 224.469,A -85,B 0,C 180,E1 -5692.27,E2 -5692.27} C_VEL
LIN {X 0,Y 506.158,Z 205.703,A -85,B 0,C 180,E1 -5695.035,E2 -5695.035} C_VEL
LIN {X 0,Y 505.882,Z 202.678,A -85,B 0,C 180,E1 -5695.509,E2 -5695.509} C_VEL
LIN {X 0,Y 502.84,Z 189.563,A -85,B 0,C 180,E1 -5697.748,E2 -5697.748} C_VEL
LIN {X 0,Y 502.808,Z 189.47,A -85,B 0,C 180,E1 -5700.21,E2 -5700.21} C_VEL
LIN {X 0,Y 502.83,Z 189.464,A -85,B 0,C 180,E1 -5703.03,E2 -5703.03} C_VEL
LIN {X 0,Y 502.78,Z 189.481,A -85,B 0,C 180,E1 -5705.95,E2 -5705.95} C_VEL
LIN {X 0,Y 502.799,Z 189.476,A -85,B 0,C 180,E1 -5708.975,E2 -5708.975} C_VEL
LIN {X 0,Y 502.793,Z 189.475,A -85,B 0,C 180,E1 -5712.138,E2 -5712.138} C_VEL
LIN {X 0,Y 502.797,Z 189.477,A -85,B 0,C 180,E1 -5715.468,E2 -5715.468} C_VEL
LIN {X 0,Y 502.817,Z 189.476,A -85,B 0,C 180,E1 -5718.934,E2 -5718.934} C_VEL
LIN {X 0,Y 502.789,Z 189.478,A -85,B 0,C 180,E1 -5722.045,E2 -5722.045} C_VEL
LIN {X 0,Y 502.805,Z 189.473,A -85,B 0,C 180,E1 -5725.034,E2 -5725.034} C_VEL
LIN {X 0,Y 502.779,Z 189.479,A -85,B 0,C 180,E1 -5727.915,E2 -5727.915} C_VEL
LIN {X 0,Y 502.834,Z 189.469,A -85,B 0,C 180,E1 -5730.713,E2 -5730.713} C_VEL
LIN {X 0,Y 502.856,Z 189.471,A -85,B 0,C 180,E1 -5733.439,E2 -5733.439} C_VEL
LIN {X 0,Y 502.785,Z 189.475,A -85,B 0,C 180,E1 -5736.086,E2 -5736.086} C_VEL
LIN {X 0,Y 502.777,Z 189.483,A -85,B 0,C 180,E1 -5738.688,E2 -5738.688} C_VEL
LIN {X 0,Y 502.824,Z 189.476,A -85,B 0,C 180,E1 -5741.248,E2 -5741.248} C_VEL
LIN {X 0,Y 502.817,Z 189.47,A -85,B 0,C 180,E1 -5743.767,E2 -5743.767} C_VEL
LIN {X 0,Y 502.829,Z 189.474,A -85,B 0,C 180,E1 -5746.254,E2 -5746.254} C_VEL
LIN {X 0,Y 502.87,Z 189.47,A -85,B 0,C 180,E1 -5748.717,E2 -5748.717} C_VEL
LIN {X 0,Y 502.895,Z 189.463,A -85,B 0,C 180,E1 -5751.966,E2 -5751.966} C_VEL
LIN {X 0,Y 502.932,Z 189.464,A -85,B 0,C 180,E1 -5754.386,E2 -5754.386} C_VEL
LIN {X 0,Y 503.018,Z 189.446,A -85,B 0,C 180,E1 -5757.598,E2 -5757.598} C_VEL
LIN {X 0,Y 503.019,Z 189.451,A -85,B 0,C 180,E1 -5760,E2 -5760} C_VEL
LIN {X 0,Y 503.017,Z 189.454,A -85,B 0,C 180,E1 -5762.402,E2 -5762.402} C_VEL
LIN {X 0,Y 502.931,Z 189.456,A -85,B 0,C 180,E1 -5765.613,E2 -5765.613} C_VEL
LIN {X 0,Y 502.894,Z 189.469,A -85,B 0,C 180,E1 -5768.033,E2 -5768.033} C_VEL
LIN {X 0,Y 502.869,Z 189.466,A -85,B 0,C 180,E1 -5771.283,E2 -5771.283} C_VEL
LIN {X 0,Y 502.838,Z 189.471,A -85,B 0,C 180,E1 -5774.571,E2 -5774.571} C_VEL
LIN {X 0,Y 502.854,Z 189.472,A -85,B 0,C 180,E1 -5777.907,E2 -5777.907} C_VEL
LIN {X 0,Y 502.821,Z 189.472,A -85,B 0,C 180,E1 -5780.536,E2 -5780.536} C_VEL
LIN {X 0,Y 502.787,Z 189.477,A -85,B 0,C 180,E1 -5783.041,E2 -5783.041} C_VEL
LIN {X 0,Y 502.835,Z 189.468,A -85,B 0,C 180,E1 -5785.676,E2 -5785.676} C_VEL
LIN {X 0,Y 502.832,Z 189.471,A -85,B 0,C 180,E1 -5788.373,E2 -5788.373} C_VEL
LIN {X 0,Y 502.787,Z 189.478,A -85,B 0,C 180,E1 -5791.499,E2 -5791.499} C_VEL
LIN {X 0,Y 502.799,Z 189.475,A -85,B 0,C 180,E1 -5794.445,E2 -5794.445} C_VEL
LIN {X 0,Y 502.774,Z 189.479,A -85,B 0,C 180,E1 -5797.179,E2 -5797.179} C_VEL
LIN {X 0,Y 502.782,Z 189.479,A -85,B 0,C 180,E1 -5800.016,E2 -5800.016} C_VEL
LIN {X 0,Y 502.797,Z 189.472,A -85,B 0,C 180,E1 -5802.2,E2 -5802.2} C_VEL
LIN {X 0,Y 502.78,Z 189.479,A -85,B 0,C 180,E1 -5805.471,E2 -5805.471} C_VEL
LIN {X 0,Y 502.815,Z 189.469,A -85,B 0,C 180,E1 -5808.935,E2 -5808.935} C_VEL
LIN {X 0,Y 502.788,Z 189.478,A -85,B 0,C 180,E1 -5812.047,E2 -5812.047} C_VEL
LIN {X 0,Y 502.791,Z 189.468,A -85,B 0,C 180,E1 -5815.034,E2 -5815.034} C_VEL
LIN {X 0,Y 502.778,Z 189.468,A -85,B 0,C 180,E1 -5817.916,E2 -5817.916} C_VEL
LIN {X 0,Y 502.866,Z 189.629,A -85,B 0,C 180,E1 -5820.77,E2 -5820.77} C_VEL
LIN {X 0,Y 507.002,Z 205.751,A -85,B 0,C 180,E1 -5823.066,E2 -5823.066} C_VEL
LIN {X 0,Y 507.225,Z 208.84,A -85,B 0,C 180,E1 -5823.459,E2 -5823.459} C_VEL
LIN {X 0,Y 505.864,Z 239.295,A -85,B 0,C 180,E1 -5827.108,E2 -5827.108} C_VEL
LIN {X 0,Y 505.607,Z 245.069,A -85,B 0,C 180,E1 -5827.769,E2 -5827.769} C_VEL
LIN {X 0,Y 508.251,Z 261.328,A -85,B 0,C 180,E1 -5828.149,E2 -5828.149} C_VEL
LIN {X 0,Y 506.789,Z 410.468,A -85,B 0,C 180,E1 -5830.402,E2 -5830.402} C_VEL
LIN {X 0,Y 506.447,Z 425.937,A -85,B 0,C 180,E1 -5830.796,E2 -5830.796} C_VEL
LIN {X 0,Y 505.995,Z 441.585,A -85,B 0,C 180,E1 -5831.37,E2 -5831.37} C_VEL
LIN {X 0,Y 505.448,Z 456.286,A -85,B 0,C 180,E1 -5832.084,E2 -5832.084} C_VEL
LIN {X 0,Y 504.931,Z 469.705,A -85,B 0,C 180,E1 -5832.901,E2 -5832.901} C_VEL
LIN {X 0,Y 504.359,Z 483.631,A -85,B 0,C 180,E1 -5833.946,E2 -5833.946} C_VEL
LIN {X 0,Y 503.851,Z 495.774,A -85,B 0,C 180,E1 -5835.046,E2 -5835.046} C_VEL
LIN {X 0,Y 503.366,Z 507.096,A -85,B 0,C 180,E1 -5836.27,E2 -5836.27} C_VEL
LIN {X 0,Y 502.973,Z 516.639,A -85,B 0,C 180,E1 -5837.492,E2 -5837.492} C_VEL
LIN {X 0,Y 502.682,Z 525.985,A -85,B 0,C 180,E1 -5838.917,E2 -5838.917} C_VEL
LIN {X 0,Y 502.406,Z 533.724,A -85,B 0,C 180,E1 -5840.337,E2 -5840.337} C_VEL
LIN {X 0,Y 502.276,Z 540.939,A -85,B 0,C 180,E1 -5841.957,E2 -5841.957} C_VEL
LIN {X 0,Y 502.184,Z 546.601,A -85,B 0,C 180,E1 -5843.572,E2 -5843.572} C_VEL
LIN {X 0,Y 502.081,Z 550.873,A -85,B 0,C 180,E1 -5845.183,E2 -5845.183} C_VEL
LIN {X 0,Y 502.107,Z 553.868,A -85,B 0,C 180,E1 -5846.791,E2 -5846.791} C_VEL
LIN {X 0,Y 502.034,Z 555.648,A -85,B 0,C 180,E1 -5848.396,E2 -5848.396} C_VEL
LIN {X 0,Y 501.979,Z 556.255,A -85,B 0,C 180,E1 -5850,E2 -5850} C_VEL
LIN {X 0,Y 502.034,Z 555.646,A -85,B 0,C 180,E1 -5851.605,E2 -5851.605} C_VEL
LIN {X 0,Y 502.107,Z 553.862,A -85,B 0,C 180,E1 -5853.21,E2 -5853.21} C_VEL
LIN {X 0,Y 502.081,Z 550.87,A -85,B 0,C 180,E1 -5854.818,E2 -5854.818} C_VEL
LIN {X 0,Y 502.233,Z 546.606,A -85,B 0,C 180,E1 -5856.428,E2 -5856.428} C_VEL
LIN {X 0,Y 502.276,Z 540.938,A -85,B 0,C 180,E1 -5858.044,E2 -5858.044} C_VEL
LIN {X 0,Y 502.406,Z 533.715,A -85,B 0,C 180,E1 -5859.664,E2 -5859.664} C_VEL
LIN {X 0,Y 502.68,Z 525.978,A -85,B 0,C 180,E1 -5861.084,E2 -5861.084} C_VEL
LIN {X 0,Y 502.975,Z 516.637,A -85,B 0,C 180,E1 -5862.508,E2 -5862.508} C_VEL
LIN {X 0,Y 503.367,Z 507.091,A -85,B 0,C 180,E1 -5863.731,E2 -5863.731} C_VEL
LIN {X 0,Y 503.901,Z 494.758,A -85,B 0,C 180,E1 -5865.056,E2 -5865.056} C_VEL
LIN {X 0,Y 504.418,Z 482.131,A -85,B 0,C 180,E1 -5866.18,E2 -5866.18} C_VEL
LIN {X 0,Y 504.975,Z 468.143,A -85,B 0,C 180,E1 -5867.202,E2 -5867.202} C_VEL
LIN {X 0,Y 505.528,Z 454.394,A -85,B 0,C 180,E1 -5868.019,E2 -5868.019} C_VEL
LIN {X 0,Y 506.076,Z 439.69,A -85,B 0,C 180,E1 -5868.709,E2 -5868.709} C_VEL
LIN {X 0,Y 506.486,Z 424.434,A -85,B 0,C 180,E1 -5869.249,E2 -5869.249} C_VEL
LIN {X 0,Y 506.812,Z 409.061,A -85,B 0,C 180,E1 -5869.624,E2 -5869.624} C_VEL
LIN {X 0,Y 508.202,Z 261.59,A -85,B 0,C 180,E1 -5871.848,E2 -5871.848} C_VEL
LIN {X 0,Y 506.08,Z 247.898,A -85,B 0,C 180,E1 -5872.15,E2 -5872.15} C_VEL
LIN {X 0,Y 505.629,Z 244.733,A -85,B 0,C 180,E1 -5872.257,E2 -5872.257} C_VEL
LIN {X 0,Y 506.457,Z 225.02,A -85,B 0,C 180,E1 -5874.601,E2 -5874.601} C_VEL
LIN {X 0,Y 507.217,Z 207.024,A -85,B 0,C 180,E1 -5876.764,E2 -5876.764} C_VEL
LIN {X 0,Y 503.554,Z 192.359,A -85,B 0,C 180,E1 -5878.808,E2 -5878.808} C_VEL
LIN {X 0,Y 502.883,Z 189.571,A -85,B 0,C 180,E1 -5879.257,E2 -5879.257} C_VEL
LIN {X 0,Y 502.78,Z 189.468,A -85,B 0,C 180,E1 -5882.085,E2 -5882.085} C_VEL
LIN {X 0,Y 502.794,Z 189.468,A -85,B 0,C 180,E1 -5884.966,E2 -5884.966} C_VEL
LIN {X 0,Y 502.791,Z 189.478,A -85,B 0,C 180,E1 -5887.954,E2 -5887.954} C_VEL
LIN {X 0,Y 502.818,Z 189.469,A -85,B 0,C 180,E1 -5891.066,E2 -5891.066} C_VEL
LIN {X 0,Y 502.783,Z 189.479,A -85,B 0,C 180,E1 -5894.53,E2 -5894.53} C_VEL
LIN {X 0,Y 502.792,Z 189.473,A -85,B 0,C 180,E1 -5897.86,E2 -5897.86} C_VEL
LIN {X 0,Y 502.799,Z 189.476,A -85,B 0,C 180,E1 -5901.024,E2 -5901.024} C_VEL
LIN {X 0,Y 502.772,Z 189.481,A -85,B 0,C 180,E1 -5904.169,E2 -5904.169} C_VEL
LIN {X 0,Y 502.83,Z 189.464,A -85,B 0,C 180,E1 -5906.993,E2 -5906.993} C_VEL
LIN {X 0,Y 502.812,Z 189.477,A -85,B 0,C 180,E1 -5910.065,E2 -5910.065} C_VEL
LIN {X 0,Y 502.827,Z 189.466,A -85,B 0,C 180,E1 -5912.533,E2 -5912.533} C_VEL
LIN {X 0,Y 502.8,Z 189.472,A -85,B 0,C 180,E1 -5915.305,E2 -5915.305} C_VEL
LIN {X 0,Y 502.777,Z 189.482,A -85,B 0,C 180,E1 -5917.826,E2 -5917.826} C_VEL
LIN {X 0,Y 502.822,Z 189.476,A -85,B 0,C 180,E1 -5920.4,E2 -5920.4} C_VEL
LIN {X 0,Y 502.828,Z 189.47,A -85,B 0,C 180,E1 -5922.932,E2 -5922.932} C_VEL
LIN {X 0,Y 502.842,Z 189.471,A -85,B 0,C 180,E1 -5925.429,E2 -5925.429} C_VEL
LIN {X 0,Y 502.874,Z 189.466,A -85,B 0,C 180,E1 -5928.717,E2 -5928.717} C_VEL
LIN {X 0,Y 502.898,Z 189.469,A -85,B 0,C 180,E1 -5931.967,E2 -5931.967} C_VEL
LIN {X 0,Y 502.934,Z 189.456,A -85,B 0,C 180,E1 -5934.387,E2 -5934.387} C_VEL
LIN {X 0,Y 503.021,Z 189.455,A -85,B 0,C 180,E1 -5937.598,E2 -5937.598} C_VEL
LIN {X 0,Y 503.024,Z 189.45,A -85,B 0,C 180,E1 -5940,E2 -5940} C_VEL
LIN {X 0,Y 503.022,Z 189.445,A -85,B 0,C 180,E1 -5942.402,E2 -5942.402} C_VEL
LIN {X 0,Y 502.935,Z 189.464,A -85,B 0,C 180,E1 -5945.614,E2 -5945.614} C_VEL
LIN {X 0,Y 502.899,Z 189.462,A -85,B 0,C 180,E1 -5948.034,E2 -5948.034} C_VEL
LIN {X 0,Y 502.874,Z 189.47,A -85,B 0,C 180,E1 -5951.283,E2 -5951.283} C_VEL
LIN {X 0,Y 502.843,Z 189.47,A -85,B 0,C 180,E1 -5954.571,E2 -5954.571} C_VEL
LIN {X 0,Y 502.853,Z 189.469,A -85,B 0,C 180,E1 -5957.907,E2 -5957.907} C_VEL
LIN {X 0,Y 502.827,Z 189.47,A -85,B 0,C 180,E1 -5960.536,E2 -5960.536} C_VEL
LIN {X 0,Y 502.789,Z 189.482,A -85,B 0,C 180,E1 -5963.041,E2 -5963.041} C_VEL
LIN {X 0,Y 502.838,Z 189.471,A -85,B 0,C 180,E1 -5965.676,E2 -5965.676} C_VEL
LIN {X 0,Y 502.838,Z 189.465,A -85,B 0,C 180,E1 -5968.373,E2 -5968.373} C_VEL
LIN {X 0,Y 502.791,Z 189.478,A -85,B 0,C 180,E1 -5971.499,E2 -5971.499} C_VEL
LIN {X 0,Y 502.806,Z 189.473,A -85,B 0,C 180,E1 -5974.445,E2 -5974.445} C_VEL
LIN {X 0,Y 502.78,Z 189.481,A -85,B 0,C 180,E1 -5977.179,E2 -5977.179} C_VEL
LIN {X 0,Y 502.787,Z 189.471,A -85,B 0,C 180,E1 -5980.016,E2 -5980.016} C_VEL
LIN {X 0,Y 502.803,Z 189.478,A -85,B 0,C 180,E1 -5982.2,E2 -5982.2} C_VEL
LIN {X 0,Y 502.801,Z 189.475,A -85,B 0,C 180,E1 -5985.469,E2 -5985.469} C_VEL
LIN {X 0,Y 502.821,Z 189.476,A -85,B 0,C 180,E1 -5988.934,E2 -5988.934} C_VEL
LIN {X 0,Y 502.793,Z 189.48,A -85,B 0,C 180,E1 -5992.046,E2 -5992.046} C_VEL
LIN {X 0,Y 502.805,Z 189.476,A -85,B 0,C 180,E1 -5995.035,E2 -5995.035} C_VEL
LIN {X 0,Y 502.809,Z 189.466,A -85,B 0,C 180,E1 -5997.225,E2 -5997.225} C_VEL
LIN {X 0,Y 502.109,Z 189.561,A -85,B 0,C 180,E1 -5997.894,E2 -5997.894} C_VEL
LIN {X 0,Y 499.247,Z 189.92,A -85,B 0,C 180,E1 -5998.98,E2 -5998.98} C_VEL
LIN {X 0,Y 496.848,Z 190.213,A -85,B 0,C 180,E1 -5999.855,E2 -5999.855} C_VEL
LIN {X 0,Y 495.821,Z 190.339,A -85,B 0,C 180,E1 -6000.53,E2 -6000.53} C_VEL
LIN {X 0,Y 495.738,Z 190.351,A -85,B 0,C 180,E1 -6000.759,E2 -6000.759} C_VEL
LIN {X 0,Y 495.805,Z 190.559,A -85,B 0,C 180,E1 -6002.087,E2 -6002.087} C_VEL
LIN {X 0,Y 499.163,Z 204.841,A -85,B 0,C 180,E1 -6004.529,E2 -6004.529} C_VEL
LIN {X 0,Y 499.35,Z 207.985,A -85,B 0,C 180,E1 -6005.025,E2 -6005.025} C_VEL
LIN {X 0,Y 498.289,Z 231.203,A -85,B 0,C 180,E1 -6008.487,E2 -6008.487} C_VEL
LIN {X 0,Y 497.801,Z 244.48,A -85,B 0,C 180,E1 -6010.395,E2 -6010.395} C_VEL
LIN {X 0,Y 500.896,Z 260.214,A -85,B 0,C 180,E1 -6010.775,E2 -6010.775} C_VEL
LIN {X 0,Y 500.128,Z 384.946,A -85,B 0,C 180,E1 -6012.52,E2 -6012.52} C_VEL
LIN {X 0,Y 499.847,Z 398.964,A -85,B 0,C 180,E1 -6012.88,E2 -6012.88} C_VEL
LIN {X 0,Y 499.442,Z 412.717,A -85,B 0,C 180,E1 -6013.402,E2 -6013.402} C_VEL
LIN {X 0,Y 499.099,Z 423.86,A -85,B 0,C 180,E1 -6013.958,E2 -6013.958} C_VEL
LIN {X 0,Y 498.43,Z 436.833,A -85,B 0,C 180,E1 -6014.774,E2 -6014.774} C_VEL
LIN {X 0,Y 497.893,Z 448.539,A -85,B 0,C 180,E1 -6015.699,E2 -6015.699} C_VEL
LIN {X 0,Y 497.279,Z 459.217,A -85,B 0,C 180,E1 -6016.723,E2 -6016.723} C_VEL
LIN {X 0,Y 496.771,Z 469.751,A -85,B 0,C 180,E1 -6017.955,E2 -6017.955} C_VEL
LIN {X 0,Y 496.281,Z 478.453,A -85,B 0,C 180,E1 -6019.185,E2 -6019.185} C_VEL
LIN {X 0,Y 495.799,Z 486.793,A -85,B 0,C 180,E1 -6020.618,E2 -6020.618} C_VEL
LIN {X 0,Y 495.551,Z 492.658,A -85,B 0,C 180,E1 -6021.847,E2 -6021.847} C_VEL
LIN {X 0,Y 495.34,Z 498.914,A -85,B 0,C 180,E1 -6023.482,E2 -6023.482} C_VEL
LIN {X 0,Y 495.076,Z 503.607,A -85,B 0,C 180,E1 -6025.114,E2 -6025.114} C_VEL
LIN {X 0,Y 495.111,Z 506.863,A -85,B 0,C 180,E1 -6026.745,E2 -6026.745} C_VEL
LIN {X 0,Y 494.963,Z 508.808,A -85,B 0,C 180,E1 -6028.372,E2 -6028.372} C_VEL
LIN {X 0,Y 494.908,Z 509.477,A -85,B 0,C 180,E1 -6030,E2 -6030} C_VEL
LIN {X 0,Y 494.961,Z 508.887,A -85,B 0,C 180,E1 -6031.627,E2 -6031.627} C_VEL
LIN {X 0,Y 495.1,Z 507.022,A -85,B 0,C 180,E1 -6033.255,E2 -6033.255} C_VEL
LIN {X 0,Y 495.074,Z 503.834,A -85,B 0,C 180,E1 -6034.886,E2 -6034.886} C_VEL
LIN {X 0,Y 495.34,Z 499.212,A -85,B 0,C 180,E1 -6036.517,E2 -6036.517} C_VEL
LIN {X 0,Y 495.525,Z 493.048,A -85,B 0,C 180,E1 -6038.153,E2 -6038.153} C_VEL
LIN {X 0,Y 495.855,Z 486.19,A -85,B 0,C 180,E1 -6039.586,E2 -6039.586} C_VEL
LIN {X 0,Y 496.291,Z 477.716,A -85,B 0,C 180,E1 -6041.021,E2 -6041.021} C_VEL
LIN {X 0,Y 496.81,Z 467.933,A -85,B 0,C 180,E1 -6042.372,E2 -6042.372} C_VEL
LIN {X 0,Y 497.417,Z 457.132,A -85,B 0,C 180,E1 -6043.585,E2 -6043.585} C_VEL
LIN {X 0,Y 497.999,Z 445.987,A -85,B 0,C 180,E1 -6044.611,E2 -6044.611} C_VEL
LIN {X 0,Y 498.561,Z 435.205,A -85,B 0,C 180,E1 -6045.43,E2 -6045.43} C_VEL
LIN {X 0,Y 499.044,Z 423.635,A -85,B 0,C 180,E1 -6046.149,E2 -6046.149} C_VEL
LIN {X 0,Y 499.54,Z 410.824,A -85,B 0,C 180,E1 -6046.772,E2 -6046.772} C_VEL
LIN {X 0,Y 499.893,Z 396.816,A -85,B 0,C 180,E1 -6047.277,E2 -6047.277} C_VEL
LIN {X 0,Y 500.136,Z 382.748,A -85,B 0,C 180,E1 -6047.611,E2 -6047.611} C_VEL
LIN {X 0,Y 500.815,Z 260.07,A -85,B 0,C 180,E1 -6049.32,E2 -6049.32} C_VEL
LIN {X 0,Y 497.807,Z 244.607,A -85,B 0,C 180,E1 -6049.689,E2 -6049.689} C_VEL
LIN {X 0,Y 497.903,Z 240.584,A -85,B 0,C 180,E1 -6050.231,E2 -6050.231} C_VEL
LIN {X 0,Y 498.744,Z 220.237,A -85,B 0,C 180,E1 -6053.238,E2 -6053.238} C_VEL
LIN {X 0,Y 499.335,Z 206.365,A -85,B 0,C 180,E1 -6055.315,E2 -6055.315} C_VEL
LIN {X 0,Y 496.739,Z 194.396,A -85,B 0,C 180,E1 -6057.329,E2 -6057.329} C_VEL
LIN {X 0,Y 495.772,Z 190.487,A -85,B 0,C 180,E1 -6058.031,E2 -6058.031} C_VEL
LIN {X 0,Y 495.75,Z 190.353,A -85,B 0,C 180,E1 -6060.687,E2 -6060.687} C_VEL
LIN {X 0,Y 495.759,Z 190.344,A -85,B 0,C 180,E1 -6063.563,E2 -6063.563} C_VEL
LIN {X 0,Y 495.731,Z 190.355,A -85,B 0,C 180,E1 -6066.543,E2 -6066.543} C_VEL
LIN {X 0,Y 495.754,Z 190.356,A -85,B 0,C 180,E1 -6069.637,E2 -6069.637} C_VEL
LIN {X 0,Y 495.734,Z 190.352,A -85,B 0,C 180,E1 -6072.506,E2 -6072.506} C_VEL
LIN {X 0,Y 495.746,Z 190.358,A -85,B 0,C 180,E1 -6075.139,E2 -6075.139} C_VEL
LIN {X 0,Y 495.754,Z 190.355,A -85,B 0,C 180,E1 -6078.218,E2 -6078.218} C_VEL
LIN {X 0,Y 495.746,Z 190.357,A -85,B 0,C 180,E1 -6081.408,E2 -6081.408} C_VEL
LIN {X 0,Y 495.753,Z 190.35,A -85,B 0,C 180,E1 -6084.462,E2 -6084.462} C_VEL
LIN {X 0,Y 495.763,Z 190.358,A -85,B 0,C 180,E1 -6087.405,E2 -6087.405} C_VEL
LIN {X 0,Y 495.776,Z 190.345,A -85,B 0,C 180,E1 -6090.254,E2 -6090.254} C_VEL
LIN {X 0,Y 495.817,Z 190.349,A -85,B 0,C 180,E1 -6093.25,E2 -6093.25} C_VEL
LIN {X 0,Y 495.746,Z 190.352,A -85,B 0,C 180,E1 -6095.724,E2 -6095.724} C_VEL
LIN {X 0,Y 495.736,Z 190.357,A -85,B 0,C 180,E1 -6098.371,E2 -6098.371} C_VEL
LIN {X 0,Y 495.778,Z 190.355,A -85,B 0,C 180,E1 -6100.971,E2 -6100.971} C_VEL
LIN {X 0,Y 495.774,Z 190.348,A -85,B 0,C 180,E1 -6103.53,E2 -6103.53} C_VEL
LIN {X 0,Y 495.79,Z 190.349,A -85,B 0,C 180,E1 -6106.055,E2 -6106.055} C_VEL
LIN {X 0,Y 495.844,Z 190.344,A -85,B 0,C 180,E1 -6108.554,E2 -6108.554} C_VEL
LIN {X 0,Y 495.866,Z 190.338,A -85,B 0,C 180,E1 -6111.852,E2 -6111.852} C_VEL
LIN {X 0,Y 495.889,Z 190.34,A -85,B 0,C 180,E1 -6114.306,E2 -6114.306} C_VEL
LIN {X 0,Y 495.987,Z 190.321,A -85,B 0,C 180,E1 -6117.564,E2 -6117.564} C_VEL
LIN {X 0,Y 495.991,Z 190.326,A -85,B 0,C 180,E1 -6120,E2 -6120} C_VEL
LIN {X 0,Y 495.986,Z 190.33,A -85,B 0,C 180,E1 -6122.436,E2 -6122.436} C_VEL
LIN {X 0,Y 495.889,Z 190.334,A -85,B 0,C 180,E1 -6125.693,E2 -6125.693} C_VEL
LIN {X 0,Y 495.865,Z 190.347,A -85,B 0,C 180,E1 -6128.148,E2 -6128.148} C_VEL
LIN {X 0,Y 495.844,Z 190.342,A -85,B 0,C 180,E1 -6131.445,E2 -6131.445} C_VEL
LIN {X 0,Y 495.782,Z 190.349,A -85,B 0,C 180,E1 -6134.783,E2 -6134.783} C_VEL
LIN {X 0,Y 495.779,Z 190.349,A -85,B 0,C 180,E1 -6137.319,E2 -6137.319} C_VEL
LIN {X 0,Y 495.765,Z 190.359,A -85,B 0,C 180,E1 -6139.89,E2 -6139.89} C_VEL
LIN {X 0,Y 495.754,Z 190.353,A -85,B 0,C 180,E1 -6142.861,E2 -6142.861} C_VEL
LIN {X 0,Y 495.792,Z 190.34,A -85,B 0,C 180,E1 -6146.068,E2 -6146.068} C_VEL
LIN {X 0,Y 495.764,Z 190.351,A -85,B 0,C 180,E1 -6148.815,E2 -6148.815} C_VEL
LIN {X 0,Y 495.749,Z 190.35,A -85,B 0,C 180,E1 -6151.726,E2 -6151.726} C_VEL
LIN {X 0,Y 495.769,Z 190.351,A -85,B 0,C 180,E1 -6154.695,E2 -6154.695} C_VEL
LIN {X 0,Y 495.724,Z 190.355,A -85,B 0,C 180,E1 -6157.562,E2 -6157.562} C_VEL
LIN {X 0,Y 495.76,Z 190.353,A -85,B 0,C 180,E1 -6160.7,E2 -6160.7} C_VEL
LIN {X 0,Y 495.722,Z 190.358,A -85,B 0,C 180,E1 -6164.002,E2 -6164.002} C_VEL
LIN {X 0,Y 495.72,Z 190.363,A -85,B 0,C 180,E1 -6167.117,E2 -6167.117} C_VEL
LIN {X 0,Y 495.751,Z 190.335,A -85,B 0,C 180,E1 -6169.954,E2 -6169.954} C_VEL
LIN {X 0,Y 495.723,Z 190.36,A -85,B 0,C 180,E1 -6172.554,E2 -6172.554} C_VEL
LIN {X 0,Y 495.766,Z 190.346,A -85,B 0,C 180,E1 -6175.457,E2 -6175.457} C_VEL
LIN {X 0,Y 495.75,Z 190.325,A -85,B 0,C 180,E1 -6178.364,E2 -6178.364} C_VEL
LIN {X 0,Y 495.825,Z 190.473,A -85,B 0,C 180,E1 -6180.434,E2 -6180.434} C_VEL
LIN {X 0,Y 500.173,Z 207.418,A -85,B 0,C 180,E1 -6182.894,E2 -6182.894} C_VEL
LIN {X 0,Y 500.479,Z 210.488,A -85,B 0,C 180,E1 -6183.298,E2 -6183.298} C_VEL
LIN {X 0,Y 499.069,Z 239.118,A -85,B 0,C 180,E1 -6186.778,E2 -6186.778} C_VEL
LIN {X 0,Y 498.809,Z 245.15,A -85,B 0,C 180,E1 -6187.477,E2 -6187.477} C_VEL
LIN {X 0,Y 501.601,Z 261.783,A -85,B 0,C 180,E1 -6187.874,E2 -6187.874} C_VEL
LIN {X 0,Y 500.032,Z 410.067,A -85,B 0,C 180,E1 -6190.153,E2 -6190.153} C_VEL
LIN {X 0,Y 499.645,Z 425.686,A -85,B 0,C 180,E1 -6190.556,E2 -6190.556} C_VEL
LIN {X 0,Y 499.183,Z 440.563,A -85,B 0,C 180,E1 -6191.107,E2 -6191.107} C_VEL
LIN {X 0,Y 498.635,Z 455.384,A -85,B 0,C 180,E1 -6191.83,E2 -6191.83} C_VEL
LIN {X 0,Y 498.047,Z 468.876,A -85,B 0,C 180,E1 -6192.657,E2 -6192.657} C_VEL
LIN {X 0,Y 497.432,Z 482.415,A -85,B 0,C 180,E1 -6193.675,E2 -6193.675} C_VEL
LIN {X 0,Y 496.856,Z 495.11,A -85,B 0,C 180,E1 -6194.831,E2 -6194.831} C_VEL
LIN {X 0,Y 496.393,Z 506.501,A -85,B 0,C 180,E1 -6196.073,E2 -6196.073} C_VEL
LIN {X 0,Y 495.948,Z 516.081,A -85,B 0,C 180,E1 -6197.312,E2 -6197.312} C_VEL
LIN {X 0,Y 495.639,Z 525.48,A -85,B 0,C 180,E1 -6198.757,E2 -6198.757} C_VEL
LIN {X 0,Y 495.331,Z 533.264,A -85,B 0,C 180,E1 -6200.197,E2 -6200.197} C_VEL
LIN {X 0,Y 495.204,Z 540.519,A -85,B 0,C 180,E1 -6201.841,E2 -6201.841} C_VEL
LIN {X 0,Y 495.086,Z 546.452,A -85,B 0,C 180,E1 -6203.557,E2 -6203.557} C_VEL
LIN {X 0,Y 495.005,Z 550.511,A -85,B 0,C 180,E1 -6205.114,E2 -6205.114} C_VEL
LIN {X 0,Y 495.027,Z 553.524,A -85,B 0,C 180,E1 -6206.745,E2 -6206.745} C_VEL
LIN {X 0,Y 494.961,Z 555.314,A -85,B 0,C 180,E1 -6208.373,E2 -6208.373} C_VEL
LIN {X 0,Y 494.897,Z 555.923,A -85,B 0,C 180,E1 -6210,E2 -6210} C_VEL
LIN {X 0,Y 494.961,Z 555.311,A -85,B 0,C 180,E1 -6211.628,E2 -6211.628} C_VEL
LIN {X 0,Y 495.027,Z 553.518,A -85,B 0,C 180,E1 -6213.256,E2 -6213.256} C_VEL
LIN {X 0,Y 495.006,Z 550.507,A -85,B 0,C 180,E1 -6214.887,E2 -6214.887} C_VEL
LIN {X 0,Y 495.162,Z 546.219,A -85,B 0,C 180,E1 -6216.52,E2 -6216.52} C_VEL
LIN {X 0,Y 495.204,Z 540.517,A -85,B 0,C 180,E1 -6218.159,E2 -6218.159} C_VEL
LIN {X 0,Y 495.331,Z 533.255,A -85,B 0,C 180,E1 -6219.803,E2 -6219.803} C_VEL
LIN {X 0,Y 495.638,Z 525.473,A -85,B 0,C 180,E1 -6221.243,E2 -6221.243} C_VEL
LIN {X 0,Y 495.949,Z 516.078,A -85,B 0,C 180,E1 -6222.688,E2 -6222.688} C_VEL
LIN {X 0,Y 496.395,Z 506.497,A -85,B 0,C 180,E1 -6223.927,E2 -6223.927} C_VEL
LIN {X 0,Y 496.896,Z 495.114,A -85,B 0,C 180,E1 -6225.169,E2 -6225.169} C_VEL
LIN {X 0,Y 497.454,Z 482.435,A -85,B 0,C 180,E1 -6226.324,E2 -6226.324} C_VEL
LIN {X 0,Y 498.02,Z 468.863,A -85,B 0,C 180,E1 -6227.344,E2 -6227.344} C_VEL
LIN {X 0,Y 498.606,Z 455.363,A -85,B 0,C 180,E1 -6228.171,E2 -6228.171} C_VEL
LIN {X 0,Y 499.204,Z 440.561,A -85,B 0,C 180,E1 -6228.893,E2 -6228.893} C_VEL
LIN {X 0,Y 499.666,Z 424.608,A -85,B 0,C 180,E1 -6229.477,E2 -6229.477} C_VEL
LIN {X 0,Y 500.037,Z 410.037,A -85,B 0,C 180,E1 -6229.847,E2 -6229.847} C_VEL
LIN {X 0,Y 501.546,Z 262.529,A -85,B 0,C 180,E1 -6232.116,E2 -6232.116} C_VEL
LIN {X 0,Y 499.793,Z 250.656,A -85,B 0,C 180,E1 -6232.378,E2 -6232.378} C_VEL
LIN {X 0,Y 498.821,Z 244.937,A -85,B 0,C 180,E1 -6232.536,E2 -6232.536} C_VEL
LIN {X 0,Y 499.722,Z 224.861,A -85,B 0,C 180,E1 -6234.955,E2 -6234.955} C_VEL
LIN {X 0,Y 500.471,Z 208.941,A -85,B 0,C 180,E1 -6236.896,E2 -6236.896} C_VEL
LIN {X 0,Y 496.796,Z 194.222,A -85,B 0,C 180,E1 -6238.981,E2 -6238.981} C_VEL
LIN {X 0,Y 495.827,Z 190.478,A -85,B 0,C 180,E1 -6239.567,E2 -6239.567} C_VEL
LIN {X 0,Y 495.75,Z 190.352,A -85,B 0,C 180,E1 -6242.595,E2 -6242.595} C_VEL
LIN {X 0,Y 495.745,Z 190.346,A -85,B 0,C 180,E1 -6245.538,E2 -6245.538} C_VEL
LIN {X 0,Y 495.758,Z 190.344,A -85,B 0,C 180,E1 -6248.768,E2 -6248.768} C_VEL
LIN {X 0,Y 495.754,Z 190.353,A -85,B 0,C 180,E1 -6251.781,E2 -6251.781} C_VEL
LIN {X 0,Y 495.735,Z 190.359,A -85,B 0,C 180,E1 -6255.141,E2 -6255.141} C_VEL
LIN {X 0,Y 495.753,Z 190.351,A -85,B 0,C 180,E1 -6258.219,E2 -6258.219} C_VEL
LIN {X 0,Y 495.748,Z 190.352,A -85,B 0,C 180,E1 -6261.408,E2 -6261.408} C_VEL
LIN {X 0,Y 495.746,Z 190.361,A -85,B 0,C 180,E1 -6264.462,E2 -6264.462} C_VEL
LIN {X 0,Y 495.765,Z 190.342,A -85,B 0,C 180,E1 -6267.406,E2 -6267.406} C_VEL
LIN {X 0,Y 495.763,Z 190.358,A -85,B 0,C 180,E1 -6270.254,E2 -6270.254} C_VEL
LIN {X 0,Y 495.82,Z 190.333,A -85,B 0,C 180,E1 -6273.251,E2 -6273.251} C_VEL
LIN {X 0,Y 495.74,Z 190.358,A -85,B 0,C 180,E1 -6276.612,E2 -6276.612} C_VEL
LIN {X 0,Y 495.775,Z 190.349,A -85,B 0,C 180,E1 -6279.324,E2 -6279.324} C_VEL
LIN {X 0,Y 495.795,Z 190.352,A -85,B 0,C 180,E1 -6281.829,E2 -6281.829} C_VEL
LIN {X 0,Y 495.787,Z 190.348,A -85,B 0,C 180,E1 -6285.217,E2 -6285.217} C_VEL
LIN {X 0,Y 495.848,Z 190.342,A -85,B 0,C 180,E1 -6288.555,E2 -6288.555} C_VEL
LIN {X 0,Y 495.87,Z 190.345,A -85,B 0,C 180,E1 -6291.852,E2 -6291.852} C_VEL
LIN {X 0,Y 495.892,Z 190.334,A -85,B 0,C 180,E1 -6294.307,E2 -6294.307} C_VEL
LIN {X 0,Y 495.989,Z 190.33,A -85,B 0,C 180,E1 -6297.564,E2 -6297.564} C_VEL
LIN {X 0,Y 495.996,Z 190.326,A -85,B 0,C 180,E1 -6300,E2 -6300} C_VEL
LIN {X 0,Y 495.99,Z 190.321,A -85,B 0,C 180,E1 -6302.436,E2 -6302.436} C_VEL
LIN {X 0,Y 495.893,Z 190.34,A -85,B 0,C 180,E1 -6305.694,E2 -6305.694} C_VEL
LIN {X 0,Y 495.871,Z 190.337,A -85,B 0,C 180,E1 -6308.148,E2 -6308.148} C_VEL
LIN {X 0,Y 495.849,Z 190.344,A -85,B 0,C 180,E1 -6311.445,E2 -6311.445} C_VEL
LIN {X 0,Y 495.788,Z 190.351,A -85,B 0,C 180,E1 -6314.783,E2 -6314.783} C_VEL
LIN {X 0,Y 495.78,Z 190.357,A -85,B 0,C 180,E1 -6317.319,E2 -6317.319} C_VEL
LIN {X 0,Y 495.769,Z 190.348,A -85,B 0,C 180,E1 -6319.891,E2 -6319.891} C_VEL
LIN {X 0,Y 495.758,Z 190.358,A -85,B 0,C 180,E1 -6322.861,E2 -6322.861} C_VEL
LIN {X 0,Y 495.789,Z 190.348,A -85,B 0,C 180,E1 -6326.068,E2 -6326.068} C_VEL
LIN {X 0,Y 495.77,Z 190.345,A -85,B 0,C 180,E1 -6328.815,E2 -6328.815} C_VEL
LIN {X 0,Y 495.753,Z 190.354,A -85,B 0,C 180,E1 -6331.726,E2 -6331.726} C_VEL
LIN {X 0,Y 495.776,Z 190.347,A -85,B 0,C 180,E1 -6334.696,E2 -6334.696} C_VEL
LIN {X 0,Y 495.73,Z 190.357,A -85,B 0,C 180,E1 -6337.562,E2 -6337.562} C_VEL
LIN {X 0,Y 495.765,Z 190.352,A -85,B 0,C 180,E1 -6340.7,E2 -6340.7} C_VEL
LIN {X 0,Y 495.733,Z 190.354,A -85,B 0,C 180,E1 -6344.001,E2 -6344.001} C_VEL
LIN {X 0,Y 495.726,Z 190.354,A -85,B 0,C 180,E1 -6347.117,E2 -6347.117} C_VEL
LIN {X 0,Y 495.759,Z 190.356,A -85,B 0,C 180,E1 -6349.953,E2 -6349.953} C_VEL
LIN {X 0,Y 495.729,Z 190.36,A -85,B 0,C 180,E1 -6352.553,E2 -6352.553} C_VEL
LIN {X 0,Y 495.783,Z 190.351,A -85,B 0,C 180,E1 -6355.457,E2 -6355.457} C_VEL
LIN {X 0,Y 495.757,Z 190.359,A -85,B 0,C 180,E1 -6358.364,E2 -6358.364} C_VEL
LIN {X 0,Y 495.738,Z 190.351,A -85,B 0,C 180,E1 -6360.759,E2 -6360.759} C_VEL
LIN {X 0,Y 495.495,Z 190.735,A -85,B 0,C 180,E1 -6361.207,E2 -6361.207} C_VEL
LIN {X 0,Y 494.519,Z 192.437,A -85,B 0,C 180,E1 -6361.85,E2 -6361.85} C_VEL
LIN {X 0,Y 493.253,Z 195.064,A -85,B 0,C 180,E1 -6362.451,E2 -6362.451} C_VEL
LIN {X 0,Y 491.838,Z 199.48,A -85,B 0,C 180,E1 -6363.226,E2 -6363.226} C_VEL
LIN {X 0,Y 491.621,Z 202.996,A -85,B 0,C 180,E1 -6363.801,E2 -6363.801} C_VEL
LIN {X 0,Y 491.81,Z 204.141,A -85,B 0,C 180,E1 -6363.993,E2 -6363.993} C_VEL
LIN {X 0,Y 492.575,Z 208.1,A -85,B 0,C 180,E1 -6364.657,E2 -6364.657} C_VEL
LIN {X 0,Y 491.582,Z 228.428,A -85,B 0,C 180,E1 -6367.737,E2 -6367.737} C_VEL
LIN {X 0,Y 490.94,Z 244.45,A -85,B 0,C 180,E1 -6370.084,E2 -6370.084} C_VEL
LIN {X 0,Y 494.255,Z 261.56,A -85,B 0,C 180,E1 -6370.503,E2 -6370.503} C_VEL
LIN {X 0,Y 493.439,Z 385.091,A -85,B 0,C 180,E1 -6372.249,E2 -6372.249} C_VEL
LIN {X 0,Y 493.145,Z 399.147,A -85,B 0,C 180,E1 -6372.613,E2 -6372.613} C_VEL
LIN {X 0,Y 492.782,Z 412.285,A -85,B 0,C 180,E1 -6373.113,E2 -6373.113} C_VEL
LIN {X 0,Y 492.397,Z 422.683,A -85,B 0,C 180,E1 -6373.627,E2 -6373.627} C_VEL
LIN {X 0,Y 491.819,Z 434.504,A -85,B 0,C 180,E1 -6374.352,E2 -6374.352} C_VEL
LIN {X 0,Y 491.249,Z 445.486,A -85,B 0,C 180,E1 -6375.183,E2 -6375.183} C_VEL
LIN {X 0,Y 490.621,Z 456.777,A -85,B 0,C 180,E1 -6376.223,E2 -6376.223} C_VEL
LIN {X 0,Y 490.039,Z 465.828,A -85,B 0,C 180,E1 -6377.224,E2 -6377.224} C_VEL
LIN {X 0,Y 489.565,Z 474.8,A -85,B 0,C 180,E1 -6378.406,E2 -6378.406} C_VEL
LIN {X 0,Y 489.091,Z 482.715,A -85,B 0,C 180,E1 -6379.652,E2 -6379.652} C_VEL
LIN {X 0,Y 488.715,Z 489.326,A -85,B 0,C 180,E1 -6380.898,E2 -6380.898} C_VEL
LIN {X 0,Y 488.387,Z 496.41,A -85,B 0,C 180,E1 -6382.558,E2 -6382.558} C_VEL
LIN {X 0,Y 488.186,Z 501.832,A -85,B 0,C 180,E1 -6384.216,E2 -6384.216} C_VEL
LIN {X 0,Y 488.076,Z 505.765,A -85,B 0,C 180,E1 -6385.871,E2 -6385.871} C_VEL
LIN {X 0,Y 488.001,Z 508.339,A -85,B 0,C 180,E1 -6387.524,E2 -6387.524} C_VEL
LIN {X 0,Y 487.837,Z 509.635,A -85,B 0,C 180,E1 -6389.174,E2 -6389.174} C_VEL
LIN {X 0,Y 487.837,Z 509.673,A -85,B 0,C 180,E1 -6390.825,E2 -6390.825} C_VEL
LIN {X 0,Y 487.999,Z 508.455,A -85,B 0,C 180,E1 -6392.476,E2 -6392.476} C_VEL
LIN {X 0,Y 488.076,Z 505.957,A -85,B 0,C 180,E1 -6394.128,E2 -6394.128} C_VEL
LIN {X 0,Y 488.185,Z 502.091,A -85,B 0,C 180,E1 -6395.783,E2 -6395.783} C_VEL
LIN {X 0,Y 488.354,Z 496.752,A -85,B 0,C 180,E1 -6397.441,E2 -6397.441} C_VEL
LIN {X 0,Y 488.702,Z 489.757,A -85,B 0,C 180,E1 -6399.101,E2 -6399.101} C_VEL
LIN {X 0,Y 489.116,Z 482.04,A -85,B 0,C 180,E1 -6400.556,E2 -6400.556} C_VEL
LIN {X 0,Y 489.597,Z 473.981,A -85,B 0,C 180,E1 -6401.803,E2 -6401.803} C_VEL
LIN {X 0,Y 490.131,Z 464.607,A -85,B 0,C 180,E1 -6403.012,E2 -6403.012} C_VEL
LIN {X 0,Y 490.762,Z 453.486,A -85,B 0,C 180,E1 -6404.195,E2 -6404.195} C_VEL
LIN {X 0,Y 491.413,Z 441.471,A -85,B 0,C 180,E1 -6405.235,E2 -6405.235} C_VEL
LIN {X 0,Y 492.059,Z 429.562,A -85,B 0,C 180,E1 -6406.065,E2 -6406.065} C_VEL
LIN {X 0,Y 492.613,Z 416.807,A -85,B 0,C 180,E1 -6406.77,E2 -6406.77} C_VEL
LIN {X 0,Y 493.025,Z 402.717,A -85,B 0,C 180,E1 -6407.358,E2 -6407.358} C_VEL
LIN {X 0,Y 493.389,Z 389.08,A -85,B 0,C 180,E1 -6407.753,E2 -6407.753} C_VEL
LIN {X 0,Y 493.552,Z 374.303,A -85,B 0,C 180,E1 -6408.014,E2 -6408.014} C_VEL
LIN {X 0,Y 494.203,Z 261.157,A -85,B 0,C 180,E1 -6409.596,E2 -6409.596} C_VEL
LIN {X 0,Y 490.919,Z 244.48,A -85,B 0,C 180,E1 -6410.006,E2 -6410.006} C_VEL
LIN {X 0,Y 491.61,Z 227.632,A -85,B 0,C 180,E1 -6412.483,E2 -6412.483} C_VEL
LIN {X 0,Y 492.557,Z 208.695,A -85,B 0,C 180,E1 -6415.343,E2 -6415.343} C_VEL
LIN {X 0,Y 491.501,Z 202.892,A -85,B 0,C 180,E1 -6416.312,E2 -6416.312} C_VEL
LIN {X 0,Y 488.744,Z 191.312,A -85,B 0,C 180,E1 -6418.373,E2 -6418.373} C_VEL
LIN {X 0,Y 488.691,Z 191.236,A -85,B 0,C 180,E1 -6421.179,E2 -6421.179} C_VEL
LIN {X 0,Y 488.732,Z 191.223,A -85,B 0,C 180,E1 -6424.112,E2 -6424.112} C_VEL
LIN {X 0,Y 488.68,Z 191.234,A -85,B 0,C 180,E1 -6427.158,E2 -6427.158} C_VEL
LIN {X 0,Y 488.715,Z 191.233,A -85,B 0,C 180,E1 -6430.344,E2 -6430.344} C_VEL
LIN {X 0,Y 488.684,Z 191.241,A -85,B 0,C 180,E1 -6433.654,E2 -6433.654} C_VEL
LIN {X 0,Y 488.683,Z 191.232,A -85,B 0,C 180,E1 -6436.345,E2 -6436.345} C_VEL
LIN {X 0,Y 488.729,Z 191.225,A -85,B 0,C 180,E1 -6439.676,E2 -6439.676} C_VEL
LIN {X 0,Y 488.678,Z 191.238,A -85,B 0,C 180,E1 -6442.841,E2 -6442.841} C_VEL
LIN {X 0,Y 488.73,Z 191.224,A -85,B 0,C 180,E1 -6445.887,E2 -6445.887} C_VEL
LIN {X 0,Y 488.69,Z 191.237,A -85,B 0,C 180,E1 -6448.82,E2 -6448.82} C_VEL
LIN {X 0,Y 488.741,Z 191.22,A -85,B 0,C 180,E1 -6451.671,E2 -6451.671} C_VEL
LIN {X 0,Y 488.741,Z 191.228,A -85,B 0,C 180,E1 -6454.444,E2 -6454.444} C_VEL
LIN {X 0,Y 488.718,Z 191.235,A -85,B 0,C 180,E1 -6457.153,E2 -6457.153} C_VEL
LIN {X 0,Y 488.719,Z 191.226,A -85,B 0,C 180,E1 -6459.81,E2 -6459.81} C_VEL
LIN {X 0,Y 488.729,Z 191.231,A -85,B 0,C 180,E1 -6462.423,E2 -6462.423} C_VEL
LIN {X 0,Y 488.755,Z 191.23,A -85,B 0,C 180,E1 -6464.999,E2 -6464.999} C_VEL
LIN {X 0,Y 488.798,Z 191.22,A -85,B 0,C 180,E1 -6468.387,E2 -6468.387} C_VEL
LIN {X 0,Y 488.81,Z 191.216,A -85,B 0,C 180,E1 -6471.733,E2 -6471.733} C_VEL
LIN {X 0,Y 488.848,Z 191.216,A -85,B 0,C 180,E1 -6474.224,E2 -6474.224} C_VEL
LIN {X 0,Y 488.954,Z 191.197,A -85,B 0,C 180,E1 -6477.528,E2 -6477.528} C_VEL
LIN {X 0,Y 488.948,Z 191.199,A -85,B 0,C 180,E1 -6480.823,E2 -6480.823} C_VEL
LIN {X 0,Y 488.954,Z 191.207,A -85,B 0,C 180,E1 -6482.471,E2 -6482.471} C_VEL
LIN {X 0,Y 488.848,Z 191.211,A -85,B 0,C 180,E1 -6485.776,E2 -6485.776} C_VEL
LIN {X 0,Y 488.81,Z 191.223,A -85,B 0,C 180,E1 -6488.266,E2 -6488.266} C_VEL
LIN {X 0,Y 488.798,Z 191.221,A -85,B 0,C 180,E1 -6491.612,E2 -6491.612} C_VEL
LIN {X 0,Y 488.754,Z 191.224,A -85,B 0,C 180,E1 -6495,E2 -6495} C_VEL
LIN {X 0,Y 488.747,Z 191.227,A -85,B 0,C 180,E1 -6498.442,E2 -6498.442} C_VEL
LIN {X 0,Y 488.699,Z 191.23,A -85,B 0,C 180,E1 -6501.071,E2 -6501.071} C_VEL
LIN {X 0,Y 488.686,Z 191.24,A -85,B 0,C 180,E1 -6503.746,E2 -6503.746} C_VEL
LIN {X 0,Y 488.792,Z 191.208,A -85,B 0,C 180,E1 -6506.946,E2 -6506.946} C_VEL
LIN {X 0,Y 488.702,Z 191.231,A -85,B 0,C 180,E1 -6510.363,E2 -6510.363} C_VEL
LIN {X 0,Y 488.729,Z 191.225,A -85,B 0,C 180,E1 -6513.485,E2 -6513.485} C_VEL
LIN {X 0,Y 488.681,Z 191.232,A -85,B 0,C 180,E1 -6516.356,E2 -6516.356} C_VEL
LIN {X 0,Y 488.695,Z 191.235,A -85,B 0,C 180,E1 -6519.255,E2 -6519.255} C_VEL
LIN {X 0,Y 488.7,Z 191.23,A -85,B 0,C 180,E1 -6521.6,E2 -6521.6} C_VEL
LIN {X 0,Y 488.695,Z 191.235,A -85,B 0,C 180,E1 -6524.803,E2 -6524.803} C_VEL
LIN {X 0,Y 488.686,Z 191.238,A -85,B 0,C 180,E1 -6527.475,E2 -6527.475} C_VEL
LIN {X 0,Y 488.728,Z 191.21,A -85,B 0,C 180,E1 -6529.677,E2 -6529.677} C_VEL
LIN {X 0,Y 488.674,Z 191.241,A -85,B 0,C 180,E1 -6532.842,E2 -6532.842} C_VEL
LIN {X 0,Y 488.716,Z 191.229,A -85,B 0,C 180,E1 -6535.887,E2 -6535.887} C_VEL
LIN {X 0,Y 488.684,Z 191.189,A -85,B 0,C 180,E1 -6538.821,E2 -6538.821} C_VEL
LIN {X 0,Y 488.766,Z 191.406,A -85,B 0,C 180,E1 -6540.112,E2 -6540.112} C_VEL
LIN {X 0,Y 493.079,Z 208.023,A -85,B 0,C 180,E1 -6542.567,E2 -6542.567} C_VEL
LIN {X 0,Y 493.728,Z 212.139,A -85,B 0,C 180,E1 -6543.132,E2 -6543.132} C_VEL
LIN {X 0,Y 492.313,Z 238.943,A -85,B 0,C 180,E1 -6546.44,E2 -6546.44} C_VEL
LIN {X 0,Y 492.045,Z 245.27,A -85,B 0,C 180,E1 -6547.178,E2 -6547.178} C_VEL
LIN {X 0,Y 494.937,Z 262.934,A -85,B 0,C 180,E1 -6547.601,E2 -6547.601} C_VEL
LIN {X 0,Y 493.283,Z 409.911,A -85,B 0,C 180,E1 -6549.897,E2 -6549.897} C_VEL
LIN {X 0,Y 492.856,Z 425.87,A -85,B 0,C 180,E1 -6550.319,E2 -6550.319} C_VEL
LIN {X 0,Y 492.347,Z 440.872,A -85,B 0,C 180,E1 -6550.888,E2 -6550.888} C_VEL
LIN {X 0,Y 491.811,Z 454.633,A -85,B 0,C 180,E1 -6551.569,E2 -6551.569} C_VEL
LIN {X 0,Y 491.162,Z 468.168,A -85,B 0,C 180,E1 -6552.406,E2 -6552.406} C_VEL
LIN {X 0,Y 490.499,Z 482.03,A -85,B 0,C 180,E1 -6553.461,E2 -6553.461} C_VEL
LIN {X 0,Y 489.916,Z 494.485,A -85,B 0,C 180,E1 -6554.611,E2 -6554.611} C_VEL
LIN {X 0,Y 489.385,Z 505.909,A -85,B 0,C 180,E1 -6555.87,E2 -6555.87} C_VEL
LIN {X 0,Y 488.862,Z 516.984,A -85,B 0,C 180,E1 -6557.336,E2 -6557.336} C_VEL
LIN {X 0,Y 488.536,Z 526.195,A -85,B 0,C 180,E1 -6558.802,E2 -6558.802} C_VEL
LIN {X 0,Y 488.277,Z 532.8,A -85,B 0,C 180,E1 -6560.054,E2 -6560.054} C_VEL
LIN {X 0,Y 488.109,Z 540.096,A -85,B 0,C 180,E1 -6561.722,E2 -6561.722} C_VEL
LIN {X 0,Y 488.029,Z 545.824,A -85,B 0,C 180,E1 -6563.385,E2 -6563.385} C_VEL
LIN {X 0,Y 487.931,Z 550.146,A -85,B 0,C 180,E1 -6565.043,E2 -6565.043} C_VEL
LIN {X 0,Y 487.949,Z 553.177,A -85,B 0,C 180,E1 -6566.698,E2 -6566.698} C_VEL
LIN {X 0,Y 487.89,Z 554.978,A -85,B 0,C 180,E1 -6568.349,E2 -6568.349} C_VEL
LIN {X 0,Y 487.818,Z 555.591,A -85,B 0,C 180,E1 -6570,E2 -6570} C_VEL
LIN {X 0,Y 487.89,Z 554.975,A -85,B 0,C 180,E1 -6571.651,E2 -6571.651} C_VEL
LIN {X 0,Y 487.949,Z 553.171,A -85,B 0,C 180,E1 -6573.303,E2 -6573.303} C_VEL
LIN {X 0,Y 487.933,Z 550.143,A -85,B 0,C 180,E1 -6574.958,E2 -6574.958} C_VEL
LIN {X 0,Y 488.07,Z 545.829,A -85,B 0,C 180,E1 -6576.615,E2 -6576.615} C_VEL
LIN {X 0,Y 488.109,Z 540.094,A -85,B 0,C 180,E1 -6578.279,E2 -6578.279} C_VEL
LIN {X 0,Y 488.277,Z 532.791,A -85,B 0,C 180,E1 -6579.946,E2 -6579.946} C_VEL
LIN {X 0,Y 488.608,Z 524.966,A -85,B 0,C 180,E1 -6581.407,E2 -6581.407} C_VEL
LIN {X 0,Y 488.938,Z 515.519,A -85,B 0,C 180,E1 -6582.874,E2 -6582.874} C_VEL
LIN {X 0,Y 489.388,Z 505.904,A -85,B 0,C 180,E1 -6584.131,E2 -6584.131} C_VEL
LIN {X 0,Y 489.905,Z 494.483,A -85,B 0,C 180,E1 -6585.39,E2 -6585.39} C_VEL
LIN {X 0,Y 490.509,Z 482.045,A -85,B 0,C 180,E1 -6586.538,E2 -6586.538} C_VEL
LIN {X 0,Y 491.117,Z 468.149,A -85,B 0,C 180,E1 -6587.596,E2 -6587.596} C_VEL
LIN {X 0,Y 491.773,Z 454.605,A -85,B 0,C 180,E1 -6588.433,E2 -6588.433} C_VEL
LIN {X 0,Y 492.413,Z 439.681,A -85,B 0,C 180,E1 -6589.164,E2 -6589.164} C_VEL
LIN {X 0,Y 492.905,Z 424.053,A -85,B 0,C 180,E1 -6589.738,E2 -6589.738} C_VEL
LIN {X 0,Y 493.306,Z 408.473,A -85,B 0,C 180,E1 -6590.13,E2 -6590.13} C_VEL
LIN {X 0,Y 494.898,Z 263.925,A -85,B 0,C 180,E1 -6592.383,E2 -6592.383} C_VEL
LIN {X 0,Y 493.942,Z 256.189,A -85,B 0,C 180,E1 -6592.549,E2 -6592.549} C_VEL
LIN {X 0,Y 492.028,Z 245.183,A -85,B 0,C 180,E1 -6592.824,E2 -6592.824} C_VEL
LIN {X 0,Y 492.94,Z 226.487,A -85,B 0,C 180,E1 -6595.097,E2 -6595.097} C_VEL
LIN {X 0,Y 493.637,Z 210.333,A -85,B 0,C 180,E1 -6597.103,E2 -6597.103} C_VEL
LIN {X 0,Y 489.492,Z 194.08,A -85,B 0,C 180,E1 -6599.456,E2 -6599.456} C_VEL
LIN {X 0,Y 488.765,Z 191.339,A -85,B 0,C 180,E1 -6599.919,E2 -6599.919} C_VEL
LIN {X 0,Y 488.701,Z 191.238,A -85,B 0,C 180,E1 -6603.125,E2 -6603.125} C_VEL
LIN {X 0,Y 488.676,Z 191.23,A -85,B 0,C 180,E1 -6606.132,E2 -6606.132} C_VEL
LIN {X 0,Y 488.696,Z 191.215,A -85,B 0,C 180,E1 -6609.255,E2 -6609.255} C_VEL
LIN {X 0,Y 488.705,Z 191.231,A -85,B 0,C 180,E1 -6611.6,E2 -6611.6} C_VEL
LIN {X 0,Y 488.699,Z 191.234,A -85,B 0,C 180,E1 -6614.803,E2 -6614.803} C_VEL
LIN {X 0,Y 488.689,Z 191.229,A -85,B 0,C 180,E1 -6617.474,E2 -6617.474} C_VEL
LIN {X 0,Y 488.731,Z 191.229,A -85,B 0,C 180,E1 -6619.676,E2 -6619.676} C_VEL
LIN {X 0,Y 488.676,Z 191.235,A -85,B 0,C 180,E1 -6622.841,E2 -6622.841} C_VEL
LIN {X 0,Y 488.728,Z 191.231,A -85,B 0,C 180,E1 -6625.887,E2 -6625.887} C_VEL
LIN {X 0,Y 488.689,Z 191.235,A -85,B 0,C 180,E1 -6628.82,E2 -6628.82} C_VEL
LIN {X 0,Y 488.74,Z 191.227,A -85,B 0,C 180,E1 -6631.671,E2 -6631.671} C_VEL
LIN {X 0,Y 488.75,Z 191.213,A -85,B 0,C 180,E1 -6633.528,E2 -6633.528} C_VEL
LIN {X 0,Y 488.677,Z 191.241,A -85,B 0,C 180,E1 -6636.254,E2 -6636.254} C_VEL
LIN {X 0,Y 488.743,Z 191.225,A -85,B 0,C 180,E1 -6639.176,E2 -6639.176} C_VEL
LIN {X 0,Y 488.73,Z 191.23,A -85,B 0,C 180,E1 -6642.423,E2 -6642.423} C_VEL
LIN {X 0,Y 488.759,Z 191.223,A -85,B 0,C 180,E1 -6645,E2 -6645} C_VEL
LIN {X 0,Y 488.802,Z 191.221,A -85,B 0,C 180,E1 -6648.388,E2 -6648.388} C_VEL
LIN {X 0,Y 488.814,Z 191.222,A -85,B 0,C 180,E1 -6651.734,E2 -6651.734} C_VEL
LIN {X 0,Y 488.851,Z 191.211,A -85,B 0,C 180,E1 -6654.224,E2 -6654.224} C_VEL
LIN {X 0,Y 488.957,Z 191.206,A -85,B 0,C 180,E1 -6657.529,E2 -6657.529} C_VEL
LIN {X 0,Y 488.967,Z 191.202,A -85,B 0,C 180,E1 -6660,E2 -6660} C_VEL
LIN {X 0,Y 488.958,Z 191.197,A -85,B 0,C 180,E1 -6662.472,E2 -6662.472} C_VEL
LIN {X 0,Y 488.852,Z 191.216,A -85,B 0,C 180,E1 -6665.776,E2 -6665.776} C_VEL
LIN {X 0,Y 488.815,Z 191.216,A -85,B 0,C 180,E1 -6668.267,E2 -6668.267} C_VEL
LIN {X 0,Y 488.803,Z 191.22,A -85,B 0,C 180,E1 -6671.613,E2 -6671.613} C_VEL
LIN {X 0,Y 488.76,Z 191.229,A -85,B 0,C 180,E1 -6675.001,E2 -6675.001} C_VEL
LIN {X 0,Y 488.753,Z 191.226,A -85,B 0,C 180,E1 -6678.442,E2 -6678.442} C_VEL
LIN {X 0,Y 488.705,Z 191.236,A -85,B 0,C 180,E1 -6681.071,E2 -6681.071} C_VEL
LIN {X 0,Y 488.687,Z 191.232,A -85,B 0,C 180,E1 -6683.746,E2 -6683.746} C_VEL
LIN {X 0,Y 488.79,Z 191.222,A -85,B 0,C 180,E1 -6686.944,E2 -6686.944} C_VEL
LIN {X 0,Y 488.708,Z 191.227,A -85,B 0,C 180,E1 -6690.363,E2 -6690.363} C_VEL
LIN {X 0,Y 488.735,Z 191.224,A -85,B 0,C 180,E1 -6693.485,E2 -6693.485} C_VEL
LIN {X 0,Y 488.688,Z 191.232,A -85,B 0,C 180,E1 -6696.356,E2 -6696.356} C_VEL
LIN {X 0,Y 488.7,Z 191.226,A -85,B 0,C 180,E1 -6699.255,E2 -6699.255} C_VEL
LIN {X 0,Y 488.706,Z 191.232,A -85,B 0,C 180,E1 -6701.6,E2 -6701.6} C_VEL
LIN {X 0,Y 488.712,Z 191.232,A -85,B 0,C 180,E1 -6704.802,E2 -6704.802} C_VEL
LIN {X 0,Y 488.692,Z 191.229,A -85,B 0,C 180,E1 -6707.475,E2 -6707.475} C_VEL
LIN {X 0,Y 488.734,Z 191.23,A -85,B 0,C 180,E1 -6709.677,E2 -6709.677} C_VEL
LIN {X 0,Y 488.681,Z 191.235,A -85,B 0,C 180,E1 -6712.841,E2 -6712.841} C_VEL
LIN {X 0,Y 488.734,Z 191.225,A -85,B 0,C 180,E1 -6715.888,E2 -6715.888} C_VEL
LIN {X 0,Y 488.694,Z 191.236,A -85,B 0,C 180,E1 -6718.82,E2 -6718.82} C_VEL
LIN {X 0,Y 488.762,Z 191.387,A -85,B 0,C 180,E1 -6721.76,E2 -6721.76} C_VEL
LIN {X 0,Y 491.81,Z 204.141,A -85,B 0,C 180,E1 -6723.993,E2 -6723.993} C_VEL
LIN {X 0,Y 491.916,Z 206.452,A -85,B 0,C 180,E1 -6724.361,E2 -6724.361} C_VEL
LIN {X 0,Y 491.358,Z 208.909,A -85,B 0,C 180,E1 -6724.713,E2 -6724.713} C_VEL
LIN {X 0,Y 489.069,Z 213.995,A -85,B 0,C 180,E1 -6725.376,E2 -6725.376} C_VEL
LIN {X 0,Y 485.889,Z 220.475,A -85,B 0,C 180,E1 -6726.211,E2 -6726.211} C_VEL
LIN {X 0,Y 484.998,Z 224.265,A -85,B 0,C 180,E1 -6726.754,E2 -6726.754} C_VEL
LIN {X 0,Y 484.131,Z 244.504,A -85,B 0,C 180,E1 -6729.771,E2 -6729.771} C_VEL
LIN {X 0,Y 487.616,Z 262.412,A -85,B 0,C 180,E1 -6730.215,E2 -6730.215} C_VEL
LIN {X 0,Y 486.77,Z 385.148,A -85,B 0,C 180,E1 -6731.97,E2 -6731.97} C_VEL
LIN {X 0,Y 486.435,Z 399.274,A -85,B 0,C 180,E1 -6732.338,E2 -6732.338} C_VEL
LIN {X 0,Y 486.036,Z 412.975,A -85,B 0,C 180,E1 -6732.869,E2 -6732.869} C_VEL
LIN {X 0,Y 485.647,Z 423.369,A -85,B 0,C 180,E1 -6733.393,E2 -6733.393} C_VEL
LIN {X 0,Y 484.928,Z 436.621,A -85,B 0,C 180,E1 -6734.232,E2 -6734.232} C_VEL
LIN {X 0,Y 484.328,Z 447.308,A -85,B 0,C 180,E1 -6735.074,E2 -6735.074} C_VEL
LIN {X 0,Y 483.652,Z 458.325,A -85,B 0,C 180,E1 -6736.127,E2 -6736.127} C_VEL
LIN {X 0,Y 483.005,Z 469.135,A -85,B 0,C 180,E1 -6737.393,E2 -6737.393} C_VEL
LIN {X 0,Y 482.426,Z 478.06,A -85,B 0,C 180,E1 -6738.658,E2 -6738.658} C_VEL
LIN {X 0,Y 481.922,Z 486.584,A -85,B 0,C 180,E1 -6740.133,E2 -6740.133} C_VEL
LIN {X 0,Y 481.496,Z 493.488,A -85,B 0,C 180,E1 -6741.607,E2 -6741.607} C_VEL
LIN {X 0,Y 481.222,Z 499.697,A -85,B 0,C 180,E1 -6743.29,E2 -6743.29} C_VEL
LIN {X 0,Y 481.018,Z 503.318,A -85,B 0,C 180,E1 -6744.55,E2 -6744.55} C_VEL
LIN {X 0,Y 481.013,Z 506.12,A -85,B 0,C 180,E1 -6745.81,E2 -6745.81} C_VEL
LIN {X 0,Y 480.939,Z 508.68,A -85,B 0,C 180,E1 -6747.487,E2 -6747.487} C_VEL
LIN {X 0,Y 480.762,Z 509.969,A -85,B 0,C 180,E1 -6749.162,E2 -6749.162} C_VEL
LIN {X 0,Y 480.763,Z 510.005,A -85,B 0,C 180,E1 -6750.837,E2 -6750.837} C_VEL
LIN {X 0,Y 480.937,Z 508.794,A -85,B 0,C 180,E1 -6752.512,E2 -6752.512} C_VEL
LIN {X 0,Y 480.993,Z 506.309,A -85,B 0,C 180,E1 -6754.189,E2 -6754.189} C_VEL
LIN {X 0,Y 481.14,Z 502.458,A -85,B 0,C 180,E1 -6755.868,E2 -6755.868} C_VEL
LIN {X 0,Y 481.329,Z 497.136,A -85,B 0,C 180,E1 -6757.551,E2 -6757.551} C_VEL
LIN {X 0,Y 481.698,Z 490.159,A -85,B 0,C 180,E1 -6759.235,E2 -6759.235} C_VEL
LIN {X 0,Y 482.134,Z 482.463,A -85,B 0,C 180,E1 -6760.711,E2 -6760.711} C_VEL
LIN {X 0,Y 482.668,Z 474.424,A -85,B 0,C 180,E1 -6761.975,E2 -6761.975} C_VEL
LIN {X 0,Y 483.214,Z 465.232,A -85,B 0,C 180,E1 -6763.182,E2 -6763.182} C_VEL
LIN {X 0,Y 483.81,Z 455.034,A -85,B 0,C 180,E1 -6764.296,E2 -6764.296} C_VEL
LIN {X 0,Y 484.506,Z 443.304,A -85,B 0,C 180,E1 -6765.35,E2 -6765.35} C_VEL
LIN {X 0,Y 485.176,Z 431.752,A -85,B 0,C 180,E1 -6766.191,E2 -6766.191} C_VEL
LIN {X 0,Y 485.708,Z 419.312,A -85,B 0,C 180,E1 -6766.919,E2 -6766.919} C_VEL
LIN {X 0,Y 486.256,Z 405.469,A -85,B 0,C 180,E1 -6767.537,E2 -6767.537} C_VEL
LIN {X 0,Y 486.649,Z 391.426,A -85,B 0,C 180,E1 -6767.98,E2 -6767.98} C_VEL
LIN {X 0,Y 486.873,Z 376.076,A -85,B 0,C 180,E1 -6768.27,E2 -6768.27} C_VEL
LIN {X 0,Y 487.523,Z 261.641,A -85,B 0,C 180,E1 -6769.891,E2 -6769.891} C_VEL
LIN {X 0,Y 484.128,Z 244.641,A -85,B 0,C 180,E1 -6770.315,E2 -6770.315} C_VEL
LIN {X 0,Y 484.307,Z 239.425,A -85,B 0,C 180,E1 -6771.048,E2 -6771.048} C_VEL
LIN {X 0,Y 485.394,Z 217.286,A -85,B 0,C 180,E1 -6774.414,E2 -6774.414} C_VEL
LIN {X 0,Y 485.772,Z 210.264,A -85,B 0,C 180,E1 -6775.493,E2 -6775.493} C_VEL
LIN {X 0,Y 483.541,Z 199.789,A -85,B 0,C 180,E1 -6777.299,E2 -6777.299} C_VEL
LIN {X 0,Y 481.667,Z 192.198,A -85,B 0,C 180,E1 -6778.693,E2 -6778.693} C_VEL
LIN {X 0,Y 481.644,Z 192.118,A -85,B 0,C 180,E1 -6781.688,E2 -6781.688} C_VEL
LIN {X 0,Y 481.691,Z 192.106,A -85,B 0,C 180,E1 -6784.681,E2 -6784.681} C_VEL
LIN {X 0,Y 481.654,Z 192.114,A -85,B 0,C 180,E1 -6788.007,E2 -6788.007} C_VEL
LIN {X 0,Y 481.654,Z 192.113,A -85,B 0,C 180,E1 -6791.041,E2 -6791.041} C_VEL
LIN {X 0,Y 481.656,Z 192.11,A -85,B 0,C 180,E1 -6794.457,E2 -6794.457} C_VEL
LIN {X 0,Y 481.644,Z 192.115,A -85,B 0,C 180,E1 -6797.839,E2 -6797.839} C_VEL
LIN {X 0,Y 481.657,Z 192.102,A -85,B 0,C 180,E1 -6800.653,E2 -6800.653} C_VEL
LIN {X 0,Y 481.627,Z 192.117,A -85,B 0,C 180,E1 -6803.375,E2 -6803.375} C_VEL
LIN {X 0,Y 481.704,Z 192.098,A -85,B 0,C 180,E1 -6806.329,E2 -6806.329} C_VEL
LIN {X 0,Y 481.652,Z 192.109,A -85,B 0,C 180,E1 -6809.415,E2 -6809.415} C_VEL
LIN {X 0,Y 481.695,Z 192.096,A -85,B 0,C 180,E1 -6812.168,E2 -6812.168} C_VEL
LIN {X 0,Y 481.712,Z 192.109,A -85,B 0,C 180,E1 -6814.969,E2 -6814.969} C_VEL
LIN {X 0,Y 481.643,Z 192.111,A -85,B 0,C 180,E1 -6817.704,E2 -6817.704} C_VEL
LIN {X 0,Y 481.699,Z 192.102,A -85,B 0,C 180,E1 -6820.393,E2 -6820.393} C_VEL
LIN {X 0,Y 481.686,Z 192.107,A -85,B 0,C 180,E1 -6823.034,E2 -6823.034} C_VEL
LIN {X 0,Y 481.684,Z 192.106,A -85,B 0,C 180,E1 -6825.638,E2 -6825.638} C_VEL
LIN {X 0,Y 481.744,Z 192.097,A -85,B 0,C 180,E1 -6828.215,E2 -6828.215} C_VEL
LIN {X 0,Y 481.756,Z 192.095,A -85,B 0,C 180,E1 -6831.611,E2 -6831.611} C_VEL
LIN {X 0,Y 481.809,Z 192.092,A -85,B 0,C 180,E1 -6834.139,E2 -6834.139} C_VEL
LIN {X 0,Y 481.921,Z 192.073,A -85,B 0,C 180,E1 -6837.492,E2 -6837.492} C_VEL
LIN {X 0,Y 481.899,Z 192.077,A -85,B 0,C 180,E1 -6840.835,E2 -6840.835} C_VEL
LIN {X 0,Y 481.921,Z 192.082,A -85,B 0,C 180,E1 -6842.507,E2 -6842.507} C_VEL
LIN {X 0,Y 481.809,Z 192.089,A -85,B 0,C 180,E1 -6845.86,E2 -6845.86} C_VEL
LIN {X 0,Y 481.755,Z 192.1,A -85,B 0,C 180,E1 -6848.388,E2 -6848.388} C_VEL
LIN {X 0,Y 481.743,Z 192.102,A -85,B 0,C 180,E1 -6851.785,E2 -6851.785} C_VEL
LIN {X 0,Y 481.735,Z 192.099,A -85,B 0,C 180,E1 -6855.224,E2 -6855.224} C_VEL
LIN {X 0,Y 481.705,Z 192.103,A -85,B 0,C 180,E1 -6858.722,E2 -6858.722} C_VEL
LIN {X 0,Y 481.638,Z 192.112,A -85,B 0,C 180,E1 -6861.395,E2 -6861.395} C_VEL
LIN {X 0,Y 481.67,Z 192.108,A -85,B 0,C 180,E1 -6864.113,E2 -6864.113} C_VEL
LIN {X 0,Y 481.745,Z 192.087,A -85,B 0,C 180,E1 -6867.141,E2 -6867.141} C_VEL
LIN {X 0,Y 481.671,Z 192.114,A -85,B 0,C 180,E1 -6869.741,E2 -6869.741} C_VEL
LIN {X 0,Y 481.665,Z 192.097,A -85,B 0,C 180,E1 -6872.675,E2 -6872.675} C_VEL
LIN {X 0,Y 481.635,Z 192.115,A -85,B 0,C 180,E1 -6875.71,E2 -6875.71} C_VEL
LIN {X 0,Y 481.665,Z 192.107,A -85,B 0,C 180,E1 -6878.86,E2 -6878.86} C_VEL
LIN {X 0,Y 481.646,Z 192.107,A -85,B 0,C 180,E1 -6881.913,E2 -6881.913} C_VEL
LIN {X 0,Y 481.649,Z 192.111,A -85,B 0,C 180,E1 -6884.458,E2 -6884.458} C_VEL
LIN {X 0,Y 481.642,Z 192.111,A -85,B 0,C 180,E1 -6887.84,E2 -6887.84} C_VEL
LIN {X 0,Y 481.653,Z 192.091,A -85,B 0,C 180,E1 -6890.655,E2 -6890.655} C_VEL
LIN {X 0,Y 481.623,Z 192.112,A -85,B 0,C 180,E1 -6893.377,E2 -6893.377} C_VEL
LIN {X 0,Y 481.666,Z 192.111,A -85,B 0,C 180,E1 -6896.327,E2 -6896.327} C_VEL
LIN {X 0,Y 481.687,Z 192.22,A -85,B 0,C 180,E1 -6899.733,E2 -6899.733} C_VEL
LIN {X 0,Y 483.81,Z 200.071,A -85,B 0,C 180,E1 -6900.968,E2 -6900.968} C_VEL
LIN {X 0,Y 486.818,Z 211.995,A -85,B 0,C 180,E1 -6902.719,E2 -6902.719} C_VEL
LIN {X 0,Y 486.841,Z 215.56,A -85,B 0,C 180,E1 -6903.185,E2 -6903.185} C_VEL
LIN {X 0,Y 485.471,Z 240.544,A -85,B 0,C 180,E1 -6906.314,E2 -6906.314} C_VEL
LIN {X 0,Y 485.263,Z 245.122,A -85,B 0,C 180,E1 -6906.858,E2 -6906.858} C_VEL
LIN {X 0,Y 488.267,Z 263.012,A -85,B 0,C 180,E1 -6907.303,E2 -6907.303} C_VEL
LIN {X 0,Y 486.617,Z 408.525,A -85,B 0,C 180,E1 -6909.609,E2 -6909.609} C_VEL
LIN {X 0,Y 486.136,Z 424.428,A -85,B 0,C 180,E1 -6910.018,E2 -6910.018} C_VEL
LIN {X 0,Y 485.595,Z 440.119,A -85,B 0,C 180,E1 -6910.612,E2 -6910.612} C_VEL
LIN {X 0,Y 484.981,Z 453.941,A -85,B 0,C 180,E1 -6911.3,E2 -6911.3} C_VEL
LIN {X 0,Y 484.288,Z 467.53,A -85,B 0,C 180,E1 -6912.148,E2 -6912.148} C_VEL
LIN {X 0,Y 483.63,Z 481.19,A -85,B 0,C 180,E1 -6913.196,E2 -6913.196} C_VEL
LIN {X 0,Y 482.987,Z 493.949,A -85,B 0,C 180,E1 -6914.384,E2 -6914.384} C_VEL
LIN {X 0,Y 482.389,Z 505.393,A -85,B 0,C 180,E1 -6915.661,E2 -6915.661} C_VEL
LIN {X 0,Y 481.846,Z 516.493,A -85,B 0,C 180,E1 -6917.149,E2 -6917.149} C_VEL
LIN {X 0,Y 481.501,Z 525.725,A -85,B 0,C 180,E1 -6918.636,E2 -6918.636} C_VEL
LIN {X 0,Y 481.19,Z 533.382,A -85,B 0,C 180,E1 -6920.119,E2 -6920.119} C_VEL
LIN {X 0,Y 481.034,Z 539.669,A -85,B 0,C 180,E1 -6921.599,E2 -6921.599} C_VEL
LIN {X 0,Y 480.952,Z 545.429,A -85,B 0,C 180,E1 -6923.287,E2 -6923.287} C_VEL
LIN {X 0,Y 480.858,Z 549.778,A -85,B 0,C 180,E1 -6924.969,E2 -6924.969} C_VEL
LIN {X 0,Y 480.873,Z 552.829,A -85,B 0,C 180,E1 -6926.649,E2 -6926.649} C_VEL
LIN {X 0,Y 480.821,Z 554.643,A -85,B 0,C 180,E1 -6928.325,E2 -6928.325} C_VEL
LIN {X 0,Y 480.741,Z 555.258,A -85,B 0,C 180,E1 -6930,E2 -6930} C_VEL
LIN {X 0,Y 480.821,Z 554.64,A -85,B 0,C 180,E1 -6931.675,E2 -6931.675} C_VEL
LIN {X 0,Y 480.873,Z 552.823,A -85,B 0,C 180,E1 -6933.352,E2 -6933.352} C_VEL
LIN {X 0,Y 480.861,Z 549.776,A -85,B 0,C 180,E1 -6935.031,E2 -6935.031} C_VEL
LIN {X 0,Y 480.97,Z 545.433,A -85,B 0,C 180,E1 -6936.713,E2 -6936.713} C_VEL
LIN {X 0,Y 481.035,Z 539.667,A -85,B 0,C 180,E1 -6938.401,E2 -6938.401} C_VEL
LIN {X 0,Y 481.24,Z 532.335,A -85,B 0,C 180,E1 -6940.093,E2 -6940.093} C_VEL
LIN {X 0,Y 481.572,Z 524.482,A -85,B 0,C 180,E1 -6941.576,E2 -6941.576} C_VEL
LIN {X 0,Y 481.924,Z 515.013,A -85,B 0,C 180,E1 -6943.064,E2 -6943.064} C_VEL
LIN {X 0,Y 482.394,Z 505.386,A -85,B 0,C 180,E1 -6944.34,E2 -6944.34} C_VEL
LIN {X 0,Y 482.955,Z 493.943,A -85,B 0,C 180,E1 -6945.618,E2 -6945.618} C_VEL
LIN {X 0,Y 483.633,Z 481.303,A -85,B 0,C 180,E1 -6946.794,E2 -6946.794} C_VEL
LIN {X 0,Y 484.267,Z 467.508,A -85,B 0,C 180,E1 -6947.853,E2 -6947.853} C_VEL
LIN {X 0,Y 484.98,Z 453.908,A -85,B 0,C 180,E1 -6948.701,E2 -6948.701} C_VEL
LIN {X 0,Y 485.648,Z 438.849,A -85,B 0,C 180,E1 -6949.441,E2 -6949.441} C_VEL
LIN {X 0,Y 486.182,Z 423.772,A -85,B 0,C 180,E1 -6950,E2 -6950} C_VEL
LIN {X 0,Y 486.57,Z 408.435,A -85,B 0,C 180,E1 -6950.393,E2 -6950.393} C_VEL
LIN {X 0,Y 488.184,Z 274.135,A -85,B 0,C 180,E1 -6952.519,E2 -6952.519} C_VEL
LIN {X 0,Y 488.107,Z 262.101,A -85,B 0,C 180,E1 -6952.717,E2 -6952.717} C_VEL
LIN {X 0,Y 485.228,Z 245.231,A -85,B 0,C 180,E1 -6953.135,E2 -6953.135} C_VEL
LIN {X 0,Y 486.221,Z 226.324,A -85,B 0,C 180,E1 -6955.469,E2 -6955.469} C_VEL
LIN {X 0,Y 486.926,Z 213.777,A -85,B 0,C 180,E1 -6957.043,E2 -6957.043} C_VEL
LIN {X 0,Y 486.381,Z 210.18,A -85,B 0,C 180,E1 -6957.541,E2 -6957.541} C_VEL
LIN {X 0,Y 482.156,Z 193.941,A -85,B 0,C 180,E1 -6959.949,E2 -6959.949} C_VEL
LIN {X 0,Y 481.69,Z 192.222,A -85,B 0,C 180,E1 -6960.267,E2 -6960.267} C_VEL
LIN {X 0,Y 481.674,Z 192.11,A -85,B 0,C 180,E1 -6963.729,E2 -6963.729} C_VEL
LIN {X 0,Y 481.624,Z 192.114,A -85,B 0,C 180,E1 -6966.747,E2 -6966.747} C_VEL
LIN {X 0,Y 481.674,Z 192.086,A -85,B 0,C 180,E1 -6969.94,E2 -6969.94} C_VEL
LIN {X 0,Y 481.636,Z 192.113,A -85,B 0,C 180,E1 -6973.3,E2 -6973.3} C_VEL
LIN {X 0,Y 481.652,Z 192.111,A -85,B 0,C 180,E1 -6975.641,E2 -6975.641} C_VEL
LIN {X 0,Y 481.654,Z 192.114,A -85,B 0,C 180,E1 -6978.958,E2 -6978.958} C_VEL
LIN {X 0,Y 481.652,Z 192.109,A -85,B 0,C 180,E1 -6981.993,E2 -6981.993} C_VEL
LIN {X 0,Y 481.686,Z 192.107,A -85,B 0,C 180,E1 -6985.318,E2 -6985.318} C_VEL
LIN {X 0,Y 481.642,Z 192.106,A -85,B 0,C 180,E1 -6988.312,E2 -6988.312} C_VEL
LIN {X 0,Y 481.695,Z 192.103,A -85,B 0,C 180,E1 -6991.218,E2 -6991.218} C_VEL
LIN {X 0,Y 481.686,Z 192.096,A -85,B 0,C 180,E1 -6994.042,E2 -6994.042} C_VEL
LIN {X 0,Y 481.671,Z 192.109,A -85,B 0,C 180,E1 -6996.812,E2 -6996.812} C_VEL
LIN {X 0,Y 481.693,Z 192.104,A -85,B 0,C 180,E1 -6999.503,E2 -6999.503} C_VEL
LIN {X 0,Y 481.703,Z 192.106,A -85,B 0,C 180,E1 -7002.158,E2 -7002.158} C_VEL
LIN {X 0,Y 481.74,Z 192.098,A -85,B 0,C 180,E1 -7004.776,E2 -7004.776} C_VEL
LIN {X 0,Y 481.748,Z 192.102,A -85,B 0,C 180,E1 -7008.215,E2 -7008.215} C_VEL
LIN {X 0,Y 481.759,Z 192.099,A -85,B 0,C 180,E1 -7011.612,E2 -7011.612} C_VEL
LIN {X 0,Y 481.812,Z 192.089,A -85,B 0,C 180,E1 -7014.14,E2 -7014.14} C_VEL
LIN {X 0,Y 481.924,Z 192.081,A -85,B 0,C 180,E1 -7017.493,E2 -7017.493} C_VEL
LIN {X 0,Y 481.938,Z 192.077,A -85,B 0,C 180,E1 -7020,E2 -7020} C_VEL
LIN {X 0,Y 481.925,Z 192.073,A -85,B 0,C 180,E1 -7022.508,E2 -7022.508} C_VEL
LIN {X 0,Y 481.813,Z 192.092,A -85,B 0,C 180,E1 -7025.861,E2 -7025.861} C_VEL
LIN {X 0,Y 481.76,Z 192.094,A -85,B 0,C 180,E1 -7028.388,E2 -7028.388} C_VEL
LIN {X 0,Y 481.748,Z 192.097,A -85,B 0,C 180,E1 -7031.785,E2 -7031.785} C_VEL
LIN {X 0,Y 481.74,Z 192.102,A -85,B 0,C 180,E1 -7035.224,E2 -7035.224} C_VEL
LIN {X 0,Y 481.71,Z 192.105,A -85,B 0,C 180,E1 -7038.722,E2 -7038.722} C_VEL
LIN {X 0,Y 481.644,Z 192.115,A -85,B 0,C 180,E1 -7041.395,E2 -7041.395} C_VEL
LIN {X 0,Y 481.672,Z 192.105,A -85,B 0,C 180,E1 -7044.114,E2 -7044.114} C_VEL
LIN {X 0,Y 481.745,Z 192.096,A -85,B 0,C 180,E1 -7047.139,E2 -7047.139} C_VEL
LIN {X 0,Y 481.677,Z 192.101,A -85,B 0,C 180,E1 -7049.741,E2 -7049.741} C_VEL
LIN {X 0,Y 481.671,Z 192.114,A -85,B 0,C 180,E1 -7052.674,E2 -7052.674} C_VEL
LIN {X 0,Y 481.642,Z 192.107,A -85,B 0,C 180,E1 -7055.709,E2 -7055.709} C_VEL
LIN {X 0,Y 481.67,Z 192.106,A -85,B 0,C 180,E1 -7058.859,E2 -7058.859} C_VEL
LIN {X 0,Y 481.652,Z 192.111,A -85,B 0,C 180,E1 -7061.913,E2 -7061.913} C_VEL
LIN {X 0,Y 481.66,Z 192.108,A -85,B 0,C 180,E1 -7064.458,E2 -7064.458} C_VEL
LIN {X 0,Y 481.648,Z 192.108,A -85,B 0,C 180,E1 -7067.84,E2 -7067.84} C_VEL
LIN {X 0,Y 481.68,Z 192.107,A -85,B 0,C 180,E1 -7070.652,E2 -7070.652} C_VEL
LIN {X 0,Y 481.629,Z 192.111,A -85,B 0,C 180,E1 -7073.376,E2 -7073.376} C_VEL
LIN {X 0,Y 481.711,Z 192.093,A -85,B 0,C 180,E1 -7076.33,E2 -7076.33} C_VEL
LIN {X 0,Y 481.652,Z 192.107,A -85,B 0,C 180,E1 -7079.418,E2 -7079.418} C_VEL
LIN {X 0,Y 481.7,Z 192.292,A -85,B 0,C 180,E1 -7081.442,E2 -7081.442} C_VEL
LIN {X 0,Y 485.532,Z 208.22,A -85,B 0,C 180,E1 -7084.263,E2 -7084.263} C_VEL
LIN {X 0,Y 485.662,Z 212.57,A -85,B 0,C 180,E1 -7084.958,E2 -7084.958} C_VEL
LIN {X 0,Y 484.998,Z 224.265,A -85,B 0,C 180,E1 -7086.754,E2 -7086.754} C_VEL
LIN {X 0,Y 484.222,Z 226.796,A -85,B 0,C 180,E1 -7087.105,E2 -7087.105} C_VEL
LIN {X 0,Y 478.331,Z 235.395,A -85,B 0,C 180,E1 -7088.127,E2 -7088.127} C_VEL
LIN {X 0,Y 477.563,Z 237.946,A -85,B 0,C 180,E1 -7088.484,E2 -7088.484} C_VEL
LIN {X 0,Y 477.309,Z 244.567,A -85,B 0,C 180,E1 -7089.449,E2 -7089.449} C_VEL
LIN {X 0,Y 480.995,Z 263.055,A -85,B 0,C 180,E1 -7089.917,E2 -7089.917} C_VEL
LIN {X 0,Y 480.089,Z 385.147,A -85,B 0,C 180,E1 -7091.683,E2 -7091.683} C_VEL
LIN {X 0,Y 479.742,Z 399.37,A -85,B 0,C 180,E1 -7092.055,E2 -7092.055} C_VEL
LIN {X 0,Y 479.368,Z 412.579,A -85,B 0,C 180,E1 -7092.569,E2 -7092.569} C_VEL
LIN {X 0,Y 478.891,Z 424.017,A -85,B 0,C 180,E1 -7093.151,E2 -7093.151} C_VEL
LIN {X 0,Y 478.119,Z 437.167,A -85,B 0,C 180,E1 -7094.001,E2 -7094.001} C_VEL
LIN {X 0,Y 477.423,Z 448.989,A -85,B 0,C 180,E1 -7094.962,E2 -7094.962} C_VEL
LIN {X 0,Y 476.788,Z 458.798,A -85,B 0,C 180,E1 -7095.924,E2 -7095.924} C_VEL
LIN {X 0,Y 476.083,Z 469.575,A -85,B 0,C 180,E1 -7097.207,E2 -7097.207} C_VEL
LIN {X 0,Y 475.47,Z 478.478,A -85,B 0,C 180,E1 -7098.489,E2 -7098.489} C_VEL
LIN {X 0,Y 474.905,Z 486.984,A -85,B 0,C 180,E1 -7099.986,E2 -7099.986} C_VEL
LIN {X 0,Y 474.487,Z 493.869,A -85,B 0,C 180,E1 -7101.482,E2 -7101.482} C_VEL
LIN {X 0,Y 474.18,Z 500.063,A -85,B 0,C 180,E1 -7103.19,E2 -7103.19} C_VEL
LIN {X 0,Y 473.97,Z 503.672,A -85,B 0,C 180,E1 -7104.469,E2 -7104.469} C_VEL
LIN {X 0,Y 473.932,Z 506.468,A -85,B 0,C 180,E1 -7105.748,E2 -7105.748} C_VEL
LIN {X 0,Y 473.85,Z 509.02,A -85,B 0,C 180,E1 -7107.449,E2 -7107.449} C_VEL
LIN {X 0,Y 473.691,Z 510.302,A -85,B 0,C 180,E1 -7109.15,E2 -7109.15} C_VEL
LIN {X 0,Y 473.691,Z 510.337,A -85,B 0,C 180,E1 -7110.85,E2 -7110.85} C_VEL
LIN {X 0,Y 473.847,Z 509.131,A -85,B 0,C 180,E1 -7112.55,E2 -7112.55} C_VEL
LIN {X 0,Y 473.915,Z 506.654,A -85,B 0,C 180,E1 -7114.252,E2 -7114.252} C_VEL
LIN {X 0,Y 474.092,Z 502.814,A -85,B 0,C 180,E1 -7115.956,E2 -7115.956} C_VEL
LIN {X 0,Y 474.287,Z 497.506,A -85,B 0,C 180,E1 -7117.663,E2 -7117.663} C_VEL
LIN {X 0,Y 474.673,Z 490.546,A -85,B 0,C 180,E1 -7119.373,E2 -7119.373} C_VEL
LIN {X 0,Y 475.162,Z 482.866,A -85,B 0,C 180,E1 -7120.87,E2 -7120.87} C_VEL
LIN {X 0,Y 475.723,Z 474.846,A -85,B 0,C 180,E1 -7122.152,E2 -7122.152} C_VEL
LIN {X 0,Y 476.368,Z 464.664,A -85,B 0,C 180,E1 -7123.502,E2 -7123.502} C_VEL
LIN {X 0,Y 477.157,Z 453.4,A -85,B 0,C 180,E1 -7124.718,E2 -7124.718} C_VEL
LIN {X 0,Y 477.886,Z 441.168,A -85,B 0,C 180,E1 -7125.787,E2 -7125.787} C_VEL
LIN {X 0,Y 478.634,Z 429.034,A -85,B 0,C 180,E1 -7126.638,E2 -7126.638} C_VEL
LIN {X 0,Y 479.132,Z 418.169,A -85,B 0,C 180,E1 -7127.257,E2 -7127.257} C_VEL
LIN {X 0,Y 479.587,Z 404.17,A -85,B 0,C 180,E1 -7127.87,E2 -7127.87} C_VEL
LIN {X 0,Y 480.021,Z 390.256,A -85,B 0,C 180,E1 -7128.292,E2 -7128.292} C_VEL
LIN {X 0,Y 480.205,Z 375.874,A -85,B 0,C 180,E1 -7128.561,E2 -7128.561} C_VEL
LIN {X 0,Y 480.911,Z 262.624,A -85,B 0,C 180,E1 -7130.184,E2 -7130.184} C_VEL
LIN {X 0,Y 477.283,Z 244.469,A -85,B 0,C 180,E1 -7130.651,E2 -7130.651} C_VEL
LIN {X 0,Y 478.083,Z 227.901,A -85,B 0,C 180,E1 -7133.155,E2 -7133.155} C_VEL
LIN {X 0,Y 478.97,Z 211.839,A -85,B 0,C 180,E1 -7135.648,E2 -7135.648} C_VEL
LIN {X 0,Y 476.177,Z 199.244,A -85,B 0,C 180,E1 -7137.867,E2 -7137.867} C_VEL
LIN {X 0,Y 474.63,Z 193.073,A -85,B 0,C 180,E1 -7139.029,E2 -7139.029} C_VEL
LIN {X 0,Y 474.614,Z 192.981,A -85,B 0,C 180,E1 -7142.43,E2 -7142.43} C_VEL
LIN {X 0,Y 474.617,Z 192.991,A -85,B 0,C 180,E1 -7145.469,E2 -7145.469} C_VEL
LIN {X 0,Y 474.609,Z 192.988,A -85,B 0,C 180,E1 -7148.456,E2 -7148.456} C_VEL
LIN {X 0,Y 474.625,Z 192.988,A -85,B 0,C 180,E1 -7150.958,E2 -7150.958} C_VEL
LIN {X 0,Y 474.606,Z 192.99,A -85,B 0,C 180,E1 -7154.104,E2 -7154.104} C_VEL
LIN {X 0,Y 474.611,Z 192.987,A -85,B 0,C 180,E1 -7157.065,E2 -7157.065} C_VEL
LIN {X 0,Y 474.613,Z 192.979,A -85,B 0,C 180,E1 -7160.353,E2 -7160.353} C_VEL
LIN {X 0,Y 474.589,Z 192.99,A -85,B 0,C 180,E1 -7163.676,E2 -7163.676} C_VEL
LIN {X 0,Y 474.638,Z 192.98,A -85,B 0,C 180,E1 -7166.779,E2 -7166.779} C_VEL
LIN {X 0,Y 474.608,Z 192.983,A -85,B 0,C 180,E1 -7169.77,E2 -7169.77} C_VEL
LIN {X 0,Y 474.691,Z 192.971,A -85,B 0,C 180,E1 -7172.679,E2 -7172.679} C_VEL
LIN {X 0,Y 474.653,Z 192.981,A -85,B 0,C 180,E1 -7175.507,E2 -7175.507} C_VEL
LIN {X 0,Y 474.664,Z 192.981,A -85,B 0,C 180,E1 -7179.185,E2 -7179.185} C_VEL
LIN {X 0,Y 474.651,Z 192.982,A -85,B 0,C 180,E1 -7181.884,E2 -7181.884} C_VEL
LIN {X 0,Y 474.693,Z 192.977,A -85,B 0,C 180,E1 -7184.544,E2 -7184.544} C_VEL
LIN {X 0,Y 474.697,Z 192.974,A -85,B 0,C 180,E1 -7188.037,E2 -7188.037} C_VEL
LIN {X 0,Y 474.721,Z 192.971,A -85,B 0,C 180,E1 -7191.486,E2 -7191.486} C_VEL
LIN {X 0,Y 474.772,Z 192.968,A -85,B 0,C 180,E1 -7194.052,E2 -7194.052} C_VEL
LIN {X 0,Y 474.887,Z 192.949,A -85,B 0,C 180,E1 -7197.455,E2 -7197.455} C_VEL
LIN {X 0,Y 474.904,Z 192.953,A -85,B 0,C 180,E1 -7200,E2 -7200} C_VEL
LIN {X 0,Y 474.887,Z 192.958,A -85,B 0,C 180,E1 -7202.544,E2 -7202.544} C_VEL
LIN {X 0,Y 474.772,Z 192.966,A -85,B 0,C 180,E1 -7205.948,E2 -7205.948} C_VEL
LIN {X 0,Y 474.721,Z 192.974,A -85,B 0,C 180,E1 -7208.514,E2 -7208.514} C_VEL
LIN {X 0,Y 474.696,Z 192.982,A -85,B 0,C 180,E1 -7211.962,E2 -7211.962} C_VEL
LIN {X 0,Y 474.692,Z 192.977,A -85,B 0,C 180,E1 -7215.456,E2 -7215.456} C_VEL
LIN {X 0,Y 474.657,Z 192.98,A -85,B 0,C 180,E1 -7219.01,E2 -7219.01} C_VEL
LIN {X 0,Y 474.581,Z 192.993,A -85,B 0,C 180,E1 -7221.729,E2 -7221.729} C_VEL
LIN {X 0,Y 474.652,Z 192.979,A -85,B 0,C 180,E1 -7224.493,E2 -7224.493} C_VEL
LIN {X 0,Y 474.692,Z 192.966,A -85,B 0,C 180,E1 -7227.339,E2 -7227.339} C_VEL
LIN {X 0,Y 474.597,Z 192.988,A -85,B 0,C 180,E1 -7230.81,E2 -7230.81} C_VEL
LIN {X 0,Y 474.632,Z 192.987,A -85,B 0,C 180,E1 -7233.984,E2 -7233.984} C_VEL
LIN {X 0,Y 474.568,Z 192.991,A -85,B 0,C 180,E1 -7236.9,E2 -7236.9} C_VEL
LIN {X 0,Y 474.622,Z 192.991,A -85,B 0,C 180,E1 -7239.648,E2 -7239.648} C_VEL
LIN {X 0,Y 474.6,Z 192.987,A -85,B 0,C 180,E1 -7242.936,E2 -7242.936} C_VEL
LIN {X 0,Y 474.6,Z 192.988,A -85,B 0,C 180,E1 -7245.895,E2 -7245.895} C_VEL
LIN {X 0,Y 474.623,Z 192.974,A -85,B 0,C 180,E1 -7249.041,E2 -7249.041} C_VEL
LIN {X 0,Y 474.604,Z 192.987,A -85,B 0,C 180,E1 -7251.705,E2 -7251.705} C_VEL
LIN {X 0,Y 474.618,Z 192.973,A -85,B 0,C 180,E1 -7254.726,E2 -7254.726} C_VEL
LIN {X 0,Y 474.623,Z 192.966,A -85,B 0,C 180,E1 -7257.788,E2 -7257.788} C_VEL
LIN {X 0,Y 474.621,Z 193.123,A -85,B 0,C 180,E1 -7259.384,E2 -7259.384} C_VEL
LIN {X 0,Y 477.731,Z 204.623,A -85,B 0,C 180,E1 -7261.192,E2 -7261.192} C_VEL
LIN {X 0,Y 479.999,Z 213.632,A -85,B 0,C 180,E1 -7262.535,E2 -7262.535} C_VEL
LIN {X 0,Y 480.24,Z 215.417,A -85,B 0,C 180,E1 -7262.786,E2 -7262.786} C_VEL
LIN {X 0,Y 478.628,Z 242.151,A -85,B 0,C 180,E1 -7266.185,E2 -7266.185} C_VEL
LIN {X 0,Y 478.479,Z 245.136,A -85,B 0,C 180,E1 -7266.536,E2 -7266.536} C_VEL
LIN {X 0,Y 481.674,Z 264.23,A -85,B 0,C 180,E1 -7267.018,E2 -7267.018} C_VEL
LIN {X 0,Y 479.907,Z 408.584,A -85,B 0,C 180,E1 -7269.339,E2 -7269.339} C_VEL
LIN {X 0,Y 479.393,Z 424.566,A -85,B 0,C 180,E1 -7269.76,E2 -7269.76} C_VEL
LIN {X 0,Y 478.843,Z 439.386,A -85,B 0,C 180,E1 -7270.327,E2 -7270.327} C_VEL
LIN {X 0,Y 478.179,Z 453.275,A -85,B 0,C 180,E1 -7271.024,E2 -7271.024} C_VEL
LIN {X 0,Y 477.443,Z 466.937,A -85,B 0,C 180,E1 -7271.883,E2 -7271.883} C_VEL
LIN {X 0,Y 476.801,Z 479.542,A -85,B 0,C 180,E1 -7272.855,E2 -7272.855} C_VEL
LIN {X 0,Y 476.109,Z 492.363,A -85,B 0,C 180,E1 -7274.043,E2 -7274.043} C_VEL
LIN {X 0,Y 475.485,Z 503.097,A -85,B 0,C 180,E1 -7275.229,E2 -7275.229} C_VEL
LIN {X 0,Y 475.014,Z 513.042,A -85,B 0,C 180,E1 -7276.525,E2 -7276.525} C_VEL
LIN {X 0,Y 474.466,Z 522.781,A -85,B 0,C 180,E1 -7278.032,E2 -7278.032} C_VEL
LIN {X 0,Y 474.27,Z 530.893,A -85,B 0,C 180,E1 -7279.542,E2 -7279.542} C_VEL
LIN {X 0,Y 473.993,Z 537.607,A -85,B 0,C 180,E1 -7281.044,E2 -7281.044} C_VEL
LIN {X 0,Y 473.85,Z 543.762,A -85,B 0,C 180,E1 -7282.758,E2 -7282.758} C_VEL
LIN {X 0,Y 473.793,Z 548.488,A -85,B 0,C 180,E1 -7284.467,E2 -7284.467} C_VEL
LIN {X 0,Y 473.711,Z 551.105,A -85,B 0,C 180,E1 -7285.746,E2 -7285.746} C_VEL
LIN {X 0,Y 473.756,Z 553.546,A -85,B 0,C 180,E1 -7287.45,E2 -7287.45} C_VEL
LIN {X 0,Y 473.686,Z 554.768,A -85,B 0,C 180,E1 -7289.15,E2 -7289.15} C_VEL
LIN {X 0,Y 473.686,Z 554.767,A -85,B 0,C 180,E1 -7290.85,E2 -7290.85} C_VEL
LIN {X 0,Y 473.756,Z 553.541,A -85,B 0,C 180,E1 -7292.551,E2 -7292.551} C_VEL
LIN {X 0,Y 473.711,Z 551.1,A -85,B 0,C 180,E1 -7294.254,E2 -7294.254} C_VEL
LIN {X 0,Y 473.833,Z 547.404,A -85,B 0,C 180,E1 -7295.96,E2 -7295.96} C_VEL
LIN {X 0,Y 473.893,Z 542.346,A -85,B 0,C 180,E1 -7297.671,E2 -7297.671} C_VEL
LIN {X 0,Y 474.02,Z 535.801,A -85,B 0,C 180,E1 -7299.386,E2 -7299.386} C_VEL
LIN {X 0,Y 474.341,Z 528.741,A -85,B 0,C 180,E1 -7300.889,E2 -7300.889} C_VEL
LIN {X 0,Y 474.659,Z 519.954,A -85,B 0,C 180,E1 -7302.439,E2 -7302.439} C_VEL
LIN {X 0,Y 475.165,Z 509.934,A -85,B 0,C 180,E1 -7303.907,E2 -7303.907} C_VEL
LIN {X 0,Y 475.712,Z 499.43,A -85,B 0,C 180,E1 -7305.203,E2 -7305.203} C_VEL
LIN {X 0,Y 476.358,Z 487.96,A -85,B 0,C 180,E1 -7306.393,E2 -7306.393} C_VEL
LIN {X 0,Y 477.014,Z 475.596,A -85,B 0,C 180,E1 -7307.469,E2 -7307.469} C_VEL
LIN {X 0,Y 477.745,Z 462.112,A -85,B 0,C 180,E1 -7308.438,E2 -7308.438} C_VEL
LIN {X 0,Y 478.467,Z 447.244,A -85,B 0,C 180,E1 -7309.299,E2 -7309.299} C_VEL
LIN {X 0,Y 479.162,Z 431.935,A -85,B 0,C 180,E1 -7309.978,E2 -7309.978} C_VEL
LIN {X 0,Y 479.658,Z 416.939,A -85,B 0,C 180,E1 -7310.464,E2 -7310.464} C_VEL
LIN {X 0,Y 480.012,Z 401.114,A -85,B 0,C 180,E1 -7310.797,E2 -7310.797} C_VEL
LIN {X 0,Y 481.596,Z 263.658,A -85,B 0,C 180,E1 -7312.993,E2 -7312.993} C_VEL
LIN {X 0,Y 478.474,Z 245.204,A -85,B 0,C 180,E1 -7313.458,E2 -7313.458} C_VEL
LIN {X 0,Y 479.534,Z 226.161,A -85,B 0,C 180,E1 -7315.85,E2 -7315.85} C_VEL
LIN {X 0,Y 480.174,Z 215.421,A -85,B 0,C 180,E1 -7317.218,E2 -7317.218} C_VEL
LIN {X 0,Y 478.704,Z 208.288,A -85,B 0,C 180,E1 -7318.252,E2 -7318.252} C_VEL
LIN {X 0,Y 474.691,Z 193.402,A -85,B 0,C 180,E1 -7320.539,E2 -7320.539} C_VEL
LIN {X 0,Y 474.598,Z 192.938,A -85,B 0,C 180,E1 -7320.809,E2 -7320.809} C_VEL
LIN {X 0,Y 474.619,Z 192.986,A -85,B 0,C 180,E1 -7323.981,E2 -7323.981} C_VEL
LIN {X 0,Y 474.57,Z 192.994,A -85,B 0,C 180,E1 -7326.899,E2 -7326.899} C_VEL
LIN {X 0,Y 474.614,Z 192.965,A -85,B 0,C 180,E1 -7329.646,E2 -7329.646} C_VEL
LIN {X 0,Y 474.623,Z 192.987,A -85,B 0,C 180,E1 -7332.237,E2 -7332.237} C_VEL
LIN {X 0,Y 474.615,Z 192.989,A -85,B 0,C 180,E1 -7335.298,E2 -7335.298} C_VEL
LIN {X 0,Y 474.618,Z 192.983,A -85,B 0,C 180,E1 -7338.214,E2 -7338.214} C_VEL
LIN {X 0,Y 474.642,Z 192.991,A -85,B 0,C 180,E1 -7340.454,E2 -7340.454} C_VEL
LIN {X 0,Y 474.586,Z 192.989,A -85,B 0,C 180,E1 -7343.676,E2 -7343.676} C_VEL
LIN {X 0,Y 474.64,Z 192.976,A -85,B 0,C 180,E1 -7346.78,E2 -7346.78} C_VEL
LIN {X 0,Y 474.602,Z 192.988,A -85,B 0,C 180,E1 -7349.77,E2 -7349.77} C_VEL
LIN {X 0,Y 474.695,Z 192.966,A -85,B 0,C 180,E1 -7352.68,E2 -7352.68} C_VEL
LIN {X 0,Y 474.638,Z 192.981,A -85,B 0,C 180,E1 -7355.506,E2 -7355.506} C_VEL
LIN {X 0,Y 474.667,Z 192.978,A -85,B 0,C 180,E1 -7359.185,E2 -7359.185} C_VEL
LIN {X 0,Y 474.654,Z 192.985,A -85,B 0,C 180,E1 -7361.884,E2 -7361.884} C_VEL
LIN {X 0,Y 474.697,Z 192.977,A -85,B 0,C 180,E1 -7364.544,E2 -7364.544} C_VEL
LIN {X 0,Y 474.701,Z 192.982,A -85,B 0,C 180,E1 -7368.038,E2 -7368.038} C_VEL
LIN {X 0,Y 474.725,Z 192.974,A -85,B 0,C 180,E1 -7371.487,E2 -7371.487} C_VEL
LIN {X 0,Y 474.775,Z 192.966,A -85,B 0,C 180,E1 -7374.053,E2 -7374.053} C_VEL
LIN {X 0,Y 474.89,Z 192.957,A -85,B 0,C 180,E1 -7377.456,E2 -7377.456} C_VEL
LIN {X 0,Y 474.908,Z 192.953,A -85,B 0,C 180,E1 -7380,E2 -7380} C_VEL
LIN {X 0,Y 474.891,Z 192.949,A -85,B 0,C 180,E1 -7382.545,E2 -7382.545} C_VEL
LIN {X 0,Y 474.776,Z 192.967,A -85,B 0,C 180,E1 -7385.948,E2 -7385.948} C_VEL
LIN {X 0,Y 474.726,Z 192.971,A -85,B 0,C 180,E1 -7388.514,E2 -7388.514} C_VEL
LIN {X 0,Y 474.702,Z 192.973,A -85,B 0,C 180,E1 -7391.963,E2 -7391.963} C_VEL
LIN {X 0,Y 474.698,Z 192.977,A -85,B 0,C 180,E1 -7395.456,E2 -7395.456} C_VEL
LIN {X 0,Y 474.663,Z 192.986,A -85,B 0,C 180,E1 -7399.011,E2 -7399.011} C_VEL
LIN {X 0,Y 474.586,Z 192.991,A -85,B 0,C 180,E1 -7401.729,E2 -7401.729} C_VEL
LIN {X 0,Y 474.655,Z 192.981,A -85,B 0,C 180,E1 -7404.493,E2 -7404.493} C_VEL
LIN {X 0,Y 474.679,Z 192.973,A -85,B 0,C 180,E1 -7407.335,E2 -7407.335} C_VEL
LIN {X 0,Y 474.603,Z 192.989,A -85,B 0,C 180,E1 -7410.81,E2 -7410.81} C_VEL
LIN {X 0,Y 474.638,Z 192.979,A -85,B 0,C 180,E1 -7413.984,E2 -7413.984} C_VEL
LIN {X 0,Y 474.575,Z 192.998,A -85,B 0,C 180,E1 -7416.9,E2 -7416.9} C_VEL
LIN {X 0,Y 474.617,Z 192.978,A -85,B 0,C 180,E1 -7419.646,E2 -7419.646} C_VEL
LIN {X 0,Y 474.623,Z 192.989,A -85,B 0,C 180,E1 -7422.237,E2 -7422.237} C_VEL
LIN {X 0,Y 474.621,Z 192.987,A -85,B 0,C 180,E1 -7425.297,E2 -7425.297} C_VEL
LIN {X 0,Y 474.621,Z 192.984,A -85,B 0,C 180,E1 -7428.215,E2 -7428.215} C_VEL
LIN {X 0,Y 474.645,Z 192.984,A -85,B 0,C 180,E1 -7430.454,E2 -7430.454} C_VEL
LIN {X 0,Y 474.591,Z 192.988,A -85,B 0,C 180,E1 -7433.677,E2 -7433.677} C_VEL
LIN {X 0,Y 474.644,Z 192.97,A -85,B 0,C 180,E1 -7436.78,E2 -7436.78} C_VEL
LIN {X 0,Y 474.604,Z 192.98,A -85,B 0,C 180,E1 -7439.77,E2 -7439.77} C_VEL
LIN {X 0,Y 474.645,Z 193.171,A -85,B 0,C 180,E1 -7441.106,E2 -7441.106} C_VEL
LIN {X 0,Y 478.335,Z 208.345,A -85,B 0,C 180,E1 -7443.846,E2 -7443.846} C_VEL
LIN {X 0,Y 478.946,Z 212.69,A -85,B 0,C 180,E1 -7444.583,E2 -7444.583} C_VEL
LIN {X 0,Y 477.731,Z 234.408,A -85,B 0,C 180,E1 -7447.943,E2 -7447.943} C_VEL
LIN {X 0,Y 477.563,Z 237.946,A -85,B 0,C 180,E1 -7448.484,E2 -7448.484} C_VEL
LIN {X 0,Y 477.337,Z 240.693,A -85,B 0,C 180,E1 -7448.81,E2 -7448.81} C_VEL
LIN {X 0,Y 476.693,Z 245.704,A -85,B 0,C 180,E1 -7449.165,E2 -7449.165} C_VEL
LIN {X 0,Y 475.89,Z 251.265,A -85,B 0,C 180,E1 -7449.387,E2 -7449.387} C_VEL
LIN {X 0,Y 474.868,Z 259.331,A -85,B 0,C 180,E1 -7449.555,E2 -7449.555} C_VEL
LIN {X 0,Y 474.417,Z 267.518,A -85,B 0,C 180,E1 -7449.67,E2 -7449.67} C_VEL
LIN {X 0,Y 473.44,Z 385.082,A -85,B 0,C 180,E1 -7451.388,E2 -7451.388} C_VEL
LIN {X 0,Y 473.067,Z 399.434,A -85,B 0,C 180,E1 -7451.765,E2 -7451.765} C_VEL
LIN {X 0,Y 472.62,Z 413.498,A -85,B 0,C 180,E1 -7452.324,E2 -7452.324} C_VEL
LIN {X 0,Y 472.148,Z 424.627,A -85,B 0,C 180,E1 -7452.903,E2 -7452.903} C_VEL
LIN {X 0,Y 471.34,Z 437.694,A -85,B 0,C 180,E1 -7453.765,E2 -7453.765} C_VEL
LIN {X 0,Y 470.58,Z 449.474,A -85,B 0,C 180,E1 -7454.738,E2 -7454.738} C_VEL
LIN {X 0,Y 469.908,Z 459.253,A -85,B 0,C 180,E1 -7455.713,E2 -7455.713} C_VEL
